  STRUCT
   FROM_MES_S702 : STRUCT
    STATION_MAIN : WORD ;
    DISTINCTION_LH_RH : WORD ;
    STAION_NUMBER : WORD ;
    BODY_TYPE_1ST : WORD ;
    BODY_TYPE_OPTION : WORD ;
    RBT1_STANDARD_WELD_DATA : WORD ;
    RBT2_STANDARD_WELD_DATA : WORD ;
    RBT3_STANDARD_WELD_DATA : WORD ;
    RBT4_STANDARD_WELD_DATA : WORD ;
    RBT5_STANDARD_WELD_DATA : WORD ;
    RBT6_STANDARD_WELD_DATA : WORD ;
    RBT7_STANDARD_WELD_DATA : WORD ;
    RBT8_STANDARD_WELD_DATA : WORD ;
    RBT9_STANDARD_WELD_DATA : WORD ;
    RBT10_STANDARD_WELD_DATA : WORD ;
    RBT11_STANDARD_WELD_DATA : WORD ;
    RBT12_STANDARD_WELD_DATA : WORD ;
    RBT13_STANDARD_WELD_DATA : WORD ;
    RBT14_STANDARD_WELD_DATA : WORD ;
    RBT15_STANDARD_WELD_DATA : WORD ;
    RBT16_STANDARD_WELD_DATA : WORD ;
    RBT17_STANDARD_WELD_DATA : WORD ;
    RBT18_STANDARD_WELD_DATA : WORD ;
    RBT19_STANDARD_WELD_DATA : WORD ;
    RBT20_STANDARD_WELD_DATA : WORD ;
    RBT21_STANDARD_WELD_DATA : WORD ;
    RBT22_STANDARD_WELD_DATA : WORD ;
    RBT23_STANDARD_WELD_DAT : WORD ;
    RBT24_STANDARD_WELD_DAT : WORD ;
    CHK_WORD : WORD ;
    TEST_TEMP : ARRAY  [1 .. 40 ] OF BYTE ;
   END_STRUCT ;
   FROM_MES_S703 : STRUCT
    STATION_MAIN : WORD ;
    DISTINCTION_LH_RH : WORD ;
    STAION_NUMBER : WORD ;
    BODY_TYPE_1ST : WORD ;
    BODY_TYPE_OPTION : WORD ;
    RBT1_STANDARD_WELD_DATA : WORD ;
    RBT2_STANDARD_WELD_DATA : WORD ;
    RBT3_STANDARD_WELD_DATA : WORD ;
    RBT4_STANDARD_WELD_DATA : WORD ;
    RBT5_STANDARD_WELD_DATA : WORD ;
    RBT6_STANDARD_WELD_DATA : WORD ;
    RBT7_STANDARD_WELD_DATA : WORD ;
    RBT8_STANDARD_WELD_DATA : WORD ;
    RBT9_STANDARD_WELD_DATA : WORD ;
    RBT10_STANDARD_WELD_DATA : WORD ;
    RBT11_STANDARD_WELD_DATA : WORD ;
    RBT12_STANDARD_WELD_DATA : WORD ;
    RBT13_STANDARD_WELD_DATA : WORD ;
    RBT14_STANDARD_WELD_DATA : WORD ;
    RBT15_STANDARD_WELD_DATA : WORD ;
    RBT16_STANDARD_WELD_DATA : WORD ;
    RBT17_STANDARD_WELD_DATA : WORD ;
    RBT18_STANDARD_WELD_DATA : WORD ;
    RBT19_STANDARD_WELD_DATA : WORD ;
    RBT20_STANDARD_WELD_DATA : WORD ;
    RBT21_STANDARD_WELD_DATA : WORD ;
    RBT22_STANDARD_WELD_DATA : WORD ;
    RBT23_STANDARD_WELD_DAT : WORD ;
    RBT24_STANDARD_WELD_DAT : WORD ;
    CHK_WORD : WORD ;
    TEST_TEMP : ARRAY  [1 .. 40 ] OF BYTE ;
   END_STRUCT ;
   FROM_MES_S704 : STRUCT
    STATION_MAIN : WORD ;
    DISTINCTION_LH_RH : WORD ;
    STAION_NUMBER : WORD ;
    BODY_TYPE_1ST : WORD ;
    BODY_TYPE_OPTION : WORD ;
    RBT1_STANDARD_WELD_DATA : WORD ;
    RBT2_STANDARD_WELD_DATA : WORD ;
    RBT3_STANDARD_WELD_DATA : WORD ;
    RBT4_STANDARD_WELD_DATA : WORD ;
    RBT5_STANDARD_WELD_DATA : WORD ;
    RBT6_STANDARD_WELD_DATA : WORD ;
    RBT7_STANDARD_WELD_DATA : WORD ;
    RBT8_STANDARD_WELD_DATA : WORD ;
    RBT9_STANDARD_WELD_DATA : WORD ;
    RBT10_STANDARD_WELD_DATA : WORD ;
    RBT11_STANDARD_WELD_DATA : WORD ;
    RBT12_STANDARD_WELD_DATA : WORD ;
    RBT13_STANDARD_WELD_DATA : WORD ;
    RBT14_STANDARD_WELD_DATA : WORD ;
    RBT15_STANDARD_WELD_DATA : WORD ;
    RBT16_STANDARD_WELD_DATA : WORD ;
    RBT17_STANDARD_WELD_DATA : WORD ;
    RBT18_STANDARD_WELD_DATA : WORD ;
    RBT19_STANDARD_WELD_DATA : WORD ;
    RBT20_STANDARD_WELD_DATA : WORD ;
    RBT21_STANDARD_WELD_DATA : WORD ;
    RBT22_STANDARD_WELD_DATA : WORD ;
    RBT23_STANDARD_WELD_DAT : WORD ;
    RBT24_STANDARD_WELD_DAT : WORD ;
    CHK_WORD : WORD ;
    TEST_TEMP : ARRAY  [1 .. 40 ] OF BYTE ;
   END_STRUCT ;
  END_STRUCT ;
BEGIN
   FROM_MES_S702.STATION_MAIN := W#16#0;
   FROM_MES_S702.DISTINCTION_LH_RH := W#16#0;
   FROM_MES_S702.STAION_NUMBER := W#16#0;
   FROM_MES_S702.BODY_TYPE_1ST := W#16#0;
   FROM_MES_S702.BODY_TYPE_OPTION := W#16#0;
   FROM_MES_S702.RBT1_STANDARD_WELD_DATA := W#16#0;
   FROM_MES_S702.RBT2_STANDARD_WELD_DATA := W#16#0;
   FROM_MES_S702.RBT3_STANDARD_WELD_DATA := W#16#0;
   FROM_MES_S702.RBT4_STANDARD_WELD_DATA := W#16#0;
   FROM_MES_S702.RBT5_STANDARD_WELD_DATA := W#16#0;
   FROM_MES_S702.RBT6_STANDARD_WELD_DATA := W#16#0;
   FROM_MES_S702.RBT7_STANDARD_WELD_DATA := W#16#0;
   FROM_MES_S702.RBT8_STANDARD_WELD_DATA := W#16#0;
   FROM_MES_S702.RBT9_STANDARD_WELD_DATA := W#16#0;
   FROM_MES_S702.RBT10_STANDARD_WELD_DATA := W#16#0;
   FROM_MES_S702.RBT11_STANDARD_WELD_DATA := W#16#0;
   FROM_MES_S702.RBT12_STANDARD_WELD_DATA := W#16#0;
   FROM_MES_S702.RBT13_STANDARD_WELD_DATA := W#16#0;
   FROM_MES_S702.RBT14_STANDARD_WELD_DATA := W#16#0;
   FROM_MES_S702.RBT15_STANDARD_WELD_DATA := W#16#0;
   FROM_MES_S702.RBT16_STANDARD_WELD_DATA := W#16#0;
   FROM_MES_S702.RBT17_STANDARD_WELD_DATA := W#16#0;
   FROM_MES_S702.RBT18_STANDARD_WELD_DATA := W#16#0;
   FROM_MES_S702.RBT19_STANDARD_WELD_DATA := W#16#0;
   FROM_MES_S702.RBT20_STANDARD_WELD_DATA := W#16#0;
   FROM_MES_S702.RBT21_STANDARD_WELD_DATA := W#16#0;
   FROM_MES_S702.RBT22_STANDARD_WELD_DATA := W#16#0;
   FROM_MES_S702.RBT23_STANDARD_WELD_DAT := W#16#0;
   FROM_MES_S702.RBT24_STANDARD_WELD_DAT := W#16#0;
   FROM_MES_S702.CHK_WORD := W#16#0;
   FROM_MES_S702.TEST_TEMP[1] := B#16#0;
   FROM_MES_S702.TEST_TEMP[2] := B#16#0;
   FROM_MES_S702.TEST_TEMP[3] := B#16#0;
   FROM_MES_S702.TEST_TEMP[4] := B#16#0;
   FROM_MES_S702.TEST_TEMP[5] := B#16#0;
   FROM_MES_S702.TEST_TEMP[6] := B#16#0;
   FROM_MES_S702.TEST_TEMP[7] := B#16#0;
   FROM_MES_S702.TEST_TEMP[8] := B#16#0;
   FROM_MES_S702.TEST_TEMP[9] := B#16#0;
   FROM_MES_S702.TEST_TEMP[10] := B#16#0;
   FROM_MES_S702.TEST_TEMP[11] := B#16#0;
   FROM_MES_S702.TEST_TEMP[12] := B#16#0;
   FROM_MES_S702.TEST_TEMP[13] := B#16#0;
   FROM_MES_S702.TEST_TEMP[14] := B#16#0;
   FROM_MES_S702.TEST_TEMP[15] := B#16#0;
   FROM_MES_S702.TEST_TEMP[16] := B#16#0;
   FROM_MES_S702.TEST_TEMP[17] := B#16#0;
   FROM_MES_S702.TEST_TEMP[18] := B#16#0;
   FROM_MES_S702.TEST_TEMP[19] := B#16#0;
   FROM_MES_S702.TEST_TEMP[20] := B#16#0;
   FROM_MES_S702.TEST_TEMP[21] := B#16#0;
   FROM_MES_S702.TEST_TEMP[22] := B#16#0;
   FROM_MES_S702.TEST_TEMP[23] := B#16#0;
   FROM_MES_S702.TEST_TEMP[24] := B#16#0;
   FROM_MES_S702.TEST_TEMP[25] := B#16#0;
   FROM_MES_S702.TEST_TEMP[26] := B#16#0;
   FROM_MES_S702.TEST_TEMP[27] := B#16#0;
   FROM_MES_S702.TEST_TEMP[28] := B#16#0;
   FROM_MES_S702.TEST_TEMP[29] := B#16#0;
   FROM_MES_S702.TEST_TEMP[30] := B#16#0;
   FROM_MES_S702.TEST_TEMP[31] := B#16#0;
   FROM_MES_S702.TEST_TEMP[32] := B#16#0;
   FROM_MES_S702.TEST_TEMP[33] := B#16#0;
   FROM_MES_S702.TEST_TEMP[34] := B#16#0;
   FROM_MES_S702.TEST_TEMP[35] := B#16#0;
   FROM_MES_S702.TEST_TEMP[36] := B#16#0;
   FROM_MES_S702.TEST_TEMP[37] := B#16#0;
   FROM_MES_S702.TEST_TEMP[38] := B#16#0;
   FROM_MES_S702.TEST_TEMP[39] := B#16#0;
   FROM_MES_S702.TEST_TEMP[40] := B#16#0;
   FROM_MES_S703.STATION_MAIN := W#16#0;
   FROM_MES_S703.DISTINCTION_LH_RH := W#16#0;
   FROM_MES_S703.STAION_NUMBER := W#16#0;
   FROM_MES_S703.BODY_TYPE_1ST := W#16#0;
   FROM_MES_S703.BODY_TYPE_OPTION := W#16#0;
   FROM_MES_S703.RBT1_STANDARD_WELD_DATA := W#16#0;
   FROM_MES_S703.RBT2_STANDARD_WELD_DATA := W#16#0;
   FROM_MES_S703.RBT3_STANDARD_WELD_DATA := W#16#0;
   FROM_MES_S703.RBT4_STANDARD_WELD_DATA := W#16#0;
   FROM_MES_S703.RBT5_STANDARD_WELD_DATA := W#16#0;
   FROM_MES_S703.RBT6_STANDARD_WELD_DATA := W#16#0;
   FROM_MES_S703.RBT7_STANDARD_WELD_DATA := W#16#0;
   FROM_MES_S703.RBT8_STANDARD_WELD_DATA := W#16#0;
   FROM_MES_S703.RBT9_STANDARD_WELD_DATA := W#16#0;
   FROM_MES_S703.RBT10_STANDARD_WELD_DATA := W#16#0;
   FROM_MES_S703.RBT11_STANDARD_WELD_DATA := W#16#0;
   FROM_MES_S703.RBT12_STANDARD_WELD_DATA := W#16#0;
   FROM_MES_S703.RBT13_STANDARD_WELD_DATA := W#16#0;
   FROM_MES_S703.RBT14_STANDARD_WELD_DATA := W#16#0;
   FROM_MES_S703.RBT15_STANDARD_WELD_DATA := W#16#0;
   FROM_MES_S703.RBT16_STANDARD_WELD_DATA := W#16#0;
   FROM_MES_S703.RBT17_STANDARD_WELD_DATA := W#16#0;
   FROM_MES_S703.RBT18_STANDARD_WELD_DATA := W#16#0;
   FROM_MES_S703.RBT19_STANDARD_WELD_DATA := W#16#0;
   FROM_MES_S703.RBT20_STANDARD_WELD_DATA := W#16#0;
   FROM_MES_S703.RBT21_STANDARD_WELD_DATA := W#16#0;
   FROM_MES_S703.RBT22_STANDARD_WELD_DATA := W#16#0;
   FROM_MES_S703.RBT23_STANDARD_WELD_DAT := W#16#0;
   FROM_MES_S703.RBT24_STANDARD_WELD_DAT := W#16#0;
   FROM_MES_S703.CHK_WORD := W#16#0;
   FROM_MES_S703.TEST_TEMP[1] := B#16#0;
   FROM_MES_S703.TEST_TEMP[2] := B#16#0;
   FROM_MES_S703.TEST_TEMP[3] := B#16#0;
   FROM_MES_S703.TEST_TEMP[4] := B#16#0;
   FROM_MES_S703.TEST_TEMP[5] := B#16#0;
   FROM_MES_S703.TEST_TEMP[6] := B#16#0;
   FROM_MES_S703.TEST_TEMP[7] := B#16#0;
   FROM_MES_S703.TEST_TEMP[8] := B#16#0;
   FROM_MES_S703.TEST_TEMP[9] := B#16#0;
   FROM_MES_S703.TEST_TEMP[10] := B#16#0;
   FROM_MES_S703.TEST_TEMP[11] := B#16#0;
   FROM_MES_S703.TEST_TEMP[12] := B#16#0;
   FROM_MES_S703.TEST_TEMP[13] := B#16#0;
   FROM_MES_S703.TEST_TEMP[14] := B#16#0;
   FROM_MES_S703.TEST_TEMP[15] := B#16#0;
   FROM_MES_S703.TEST_TEMP[16] := B#16#0;
   FROM_MES_S703.TEST_TEMP[17] := B#16#0;
   FROM_MES_S703.TEST_TEMP[18] := B#16#0;
   FROM_MES_S703.TEST_TEMP[19] := B#16#0;
   FROM_MES_S703.TEST_TEMP[20] := B#16#0;
   FROM_MES_S703.TEST_TEMP[21] := B#16#0;
   FROM_MES_S703.TEST_TEMP[22] := B#16#0;
   FROM_MES_S703.TEST_TEMP[23] := B#16#0;
   FROM_MES_S703.TEST_TEMP[24] := B#16#0;
   FROM_MES_S703.TEST_TEMP[25] := B#16#0;
   FROM_MES_S703.TEST_TEMP[26] := B#16#0;
   FROM_MES_S703.TEST_TEMP[27] := B#16#0;
   FROM_MES_S703.TEST_TEMP[28] := B#16#0;
   FROM_MES_S703.TEST_TEMP[29] := B#16#0;
   FROM_MES_S703.TEST_TEMP[30] := B#16#0;
   FROM_MES_S703.TEST_TEMP[31] := B#16#0;
   FROM_MES_S703.TEST_TEMP[32] := B#16#0;
   FROM_MES_S703.TEST_TEMP[33] := B#16#0;
   FROM_MES_S703.TEST_TEMP[34] := B#16#0;
   FROM_MES_S703.TEST_TEMP[35] := B#16#0;
   FROM_MES_S703.TEST_TEMP[36] := B#16#0;
   FROM_MES_S703.TEST_TEMP[37] := B#16#0;
   FROM_MES_S703.TEST_TEMP[38] := B#16#0;
   FROM_MES_S703.TEST_TEMP[39] := B#16#0;
   FROM_MES_S703.TEST_TEMP[40] := B#16#0;
   FROM_MES_S704.STATION_MAIN := W#16#0;
   FROM_MES_S704.DISTINCTION_LH_RH := W#16#0;
   FROM_MES_S704.STAION_NUMBER := W#16#0;
   FROM_MES_S704.BODY_TYPE_1ST := W#16#0;
   FROM_MES_S704.BODY_TYPE_OPTION := W#16#0;
   FROM_MES_S704.RBT1_STANDARD_WELD_DATA := W#16#0;
   FROM_MES_S704.RBT2_STANDARD_WELD_DATA := W#16#0;
   FROM_MES_S704.RBT3_STANDARD_WELD_DATA := W#16#0;
   FROM_MES_S704.RBT4_STANDARD_WELD_DATA := W#16#0;
   FROM_MES_S704.RBT5_STANDARD_WELD_DATA := W#16#0;
   FROM_MES_S704.RBT6_STANDARD_WELD_DATA := W#16#0;
   FROM_MES_S704.RBT7_STANDARD_WELD_DATA := W#16#0;
   FROM_MES_S704.RBT8_STANDARD_WELD_DATA := W#16#0;
   FROM_MES_S704.RBT9_STANDARD_WELD_DATA := W#16#0;
   FROM_MES_S704.RBT10_STANDARD_WELD_DATA := W#16#0;
   FROM_MES_S704.RBT11_STANDARD_WELD_DATA := W#16#0;
   FROM_MES_S704.RBT12_STANDARD_WELD_DATA := W#16#0;
   FROM_MES_S704.RBT13_STANDARD_WELD_DATA := W#16#0;
   FROM_MES_S704.RBT14_STANDARD_WELD_DATA := W#16#0;
   FROM_MES_S704.RBT15_STANDARD_WELD_DATA := W#16#0;
   FROM_MES_S704.RBT16_STANDARD_WELD_DATA := W#16#0;
   FROM_MES_S704.RBT17_STANDARD_WELD_DATA := W#16#0;
   FROM_MES_S704.RBT18_STANDARD_WELD_DATA := W#16#0;
   FROM_MES_S704.RBT19_STANDARD_WELD_DATA := W#16#0;
   FROM_MES_S704.RBT20_STANDARD_WELD_DATA := W#16#0;
   FROM_MES_S704.RBT21_STANDARD_WELD_DATA := W#16#0;
   FROM_MES_S704.RBT22_STANDARD_WELD_DATA := W#16#0;
   FROM_MES_S704.RBT23_STANDARD_WELD_DAT := W#16#0;
   FROM_MES_S704.RBT24_STANDARD_WELD_DAT := W#16#0;
   FROM_MES_S704.CHK_WORD := W#16#0;
   FROM_MES_S704.TEST_TEMP[1] := B#16#0;
   FROM_MES_S704.TEST_TEMP[2] := B#16#0;
   FROM_MES_S704.TEST_TEMP[3] := B#16#0;
   FROM_MES_S704.TEST_TEMP[4] := B#16#0;
   FROM_MES_S704.TEST_TEMP[5] := B#16#0;
   FROM_MES_S704.TEST_TEMP[6] := B#16#0;
   FROM_MES_S704.TEST_TEMP[7] := B#16#0;
   FROM_MES_S704.TEST_TEMP[8] := B#16#0;
   FROM_MES_S704.TEST_TEMP[9] := B#16#0;
   FROM_MES_S704.TEST_TEMP[10] := B#16#0;
   FROM_MES_S704.TEST_TEMP[11] := B#16#0;
   FROM_MES_S704.TEST_TEMP[12] := B#16#0;
   FROM_MES_S704.TEST_TEMP[13] := B#16#0;
   FROM_MES_S704.TEST_TEMP[14] := B#16#0;
   FROM_MES_S704.TEST_TEMP[15] := B#16#0;
   FROM_MES_S704.TEST_TEMP[16] := B#16#0;
   FROM_MES_S704.TEST_TEMP[17] := B#16#0;
   FROM_MES_S704.TEST_TEMP[18] := B#16#0;
   FROM_MES_S704.TEST_TEMP[19] := B#16#0;
   FROM_MES_S704.TEST_TEMP[20] := B#16#0;
   FROM_MES_S704.TEST_TEMP[21] := B#16#0;
   FROM_MES_S704.TEST_TEMP[22] := B#16#0;
   FROM_MES_S704.TEST_TEMP[23] := B#16#0;
   FROM_MES_S704.TEST_TEMP[24] := B#16#0;
   FROM_MES_S704.TEST_TEMP[25] := B#16#0;
   FROM_MES_S704.TEST_TEMP[26] := B#16#0;
   FROM_MES_S704.TEST_TEMP[27] := B#16#0;
   FROM_MES_S704.TEST_TEMP[28] := B#16#0;
   FROM_MES_S704.TEST_TEMP[29] := B#16#0;
   FROM_MES_S704.TEST_TEMP[30] := B#16#0;
   FROM_MES_S704.TEST_TEMP[31] := B#16#0;
   FROM_MES_S704.TEST_TEMP[32] := B#16#0;
   FROM_MES_S704.TEST_TEMP[33] := B#16#0;
   FROM_MES_S704.TEST_TEMP[34] := B#16#0;
   FROM_MES_S704.TEST_TEMP[35] := B#16#0;
   FROM_MES_S704.TEST_TEMP[36] := B#16#0;
   FROM_MES_S704.TEST_TEMP[37] := B#16#0;
   FROM_MES_S704.TEST_TEMP[38] := B#16#0;
   FROM_MES_S704.TEST_TEMP[39] := B#16#0;
   FROM_MES_S704.TEST_TEMP[40] := B#16#0;
END_DATA_BLOCK

DATA_BLOCK DB 41
TITLE =
VERSION : 0.1


  STRUCT
   S702_BT_CODE_2011 : STRUCT
    STATION_MAIN : WORD ;
    DISTINCTION_LH_RH : WORD ;
    STAION_NUMBER : WORD ;
    BODY_TYPE_1ST : WORD ;
    BODY_TYPE_OPTION : WORD ;
    RBT1_STANDARD_WELD_DATA : WORD ;
    RBT2_STANDARD_WELD_DATA : WORD ;
    RBT3_STANDARD_WELD_DATA : WORD ;
    RBT4_STANDARD_WELD_DATA : WORD ;
    RBT5_STANDARD_WELD_DATA : WORD ;
    RBT6_STANDARD_WELD_DATA : WORD ;
    RBT7_STANDARD_WELD_DATA : WORD ;
    RBT8_STANDARD_WELD_DATA : WORD ;
    RBT9_STANDARD_WELD_DATA : WORD ;
    RBT10_STANDARD_WELD_DATA : WORD ;
    RBT11_STANDARD_WELD_DATA : WORD ;
    RBT12_STANDARD_WELD_DATA : WORD ;
    RBT13_STANDARD_WELD_DATA : WORD ;
    RBT14_STANDARD_WELD_DATA : WORD ;
    RBT15_STANDARD_WELD_DATA : WORD ;
    RBT16_STANDARD_WELD_DATA : WORD ;
    RBT17_STANDARD_WELD_DATA : WORD ;
    RBT18_STANDARD_WELD_DATA : WORD ;
    RBT19_STANDARD_WELD_DATA : WORD ;
    RBT20_STANDARD_WELD_DATA : WORD ;
    RBT21_STANDARD_WELD_DATA : WORD ;
    RBT22_STANDARD_WELD_DATA : WORD ;
    RBT23_STANDARD_WELD_DAT : WORD ;
    RBT24_STANDARD_WELD_DAT : WORD ;
    CHK_WORD : WORD ;
    TEST_TEMP : ARRAY  [1 .. 40 ] OF BYTE ;
   END_STRUCT ;
   S702_BT_CODE_2012 : STRUCT
    STATION_MAIN : WORD ;
    DISTINCTION_LH_RH : WORD ;
    STAION_NUMBER : WORD ;
    BODY_TYPE_1ST : WORD ;
    BODY_TYPE_OPTION : WORD ;
    RBT1_STANDARD_WELD_DATA : WORD ;
    RBT2_STANDARD_WELD_DATA : WORD ;
    RBT3_STANDARD_WELD_DATA : WORD ;
    RBT4_STANDARD_WELD_DATA : WORD ;
    RBT5_STANDARD_WELD_DATA : WORD ;
    RBT6_STANDARD_WELD_DATA : WORD ;
    RBT7_STANDARD_WELD_DATA : WORD ;
    RBT8_STANDARD_WELD_DATA : WORD ;
    RBT9_STANDARD_WELD_DATA : WORD ;
    RBT10_STANDARD_WELD_DATA : WORD ;
    RBT11_STANDARD_WELD_DATA : WORD ;
    RBT12_STANDARD_WELD_DATA : WORD ;
    RBT13_STANDARD_WELD_DATA : WORD ;
    RBT14_STANDARD_WELD_DATA : WORD ;
    RBT15_STANDARD_WELD_DATA : WORD ;
    RBT16_STANDARD_WELD_DATA : WORD ;
    RBT17_STANDARD_WELD_DATA : WORD ;
    RBT18_STANDARD_WELD_DATA : WORD ;
    RBT19_STANDARD_WELD_DATA : WORD ;
    RBT20_STANDARD_WELD_DATA : WORD ;
    RBT21_STANDARD_WELD_DATA : WORD ;
    RBT22_STANDARD_WELD_DATA : WORD ;
    RBT23_STANDARD_WELD_DAT : WORD ;
    RBT24_STANDARD_WELD_DAT : WORD ;
    CHK_WORD : WORD ;
    TEST_TEMP : ARRAY  [1 .. 40 ] OF BYTE ;
   END_STRUCT ;
   S702_BT_CODE_2013 : STRUCT
    STATION_MAIN : WORD ;
    DISTINCTION_LH_RH : WORD ;
    STAION_NUMBER : WORD ;
    BODY_TYPE_1ST : WORD ;
    BODY_TYPE_OPTION : WORD ;
    RBT1_STANDARD_WELD_DATA : WORD ;
    RBT2_STANDARD_WELD_DATA : WORD ;
    RBT3_STANDARD_WELD_DATA : WORD ;
    RBT4_STANDARD_WELD_DATA : WORD ;
    RBT5_STANDARD_WELD_DATA : WORD ;
    RBT6_STANDARD_WELD_DATA : WORD ;
    RBT7_STANDARD_WELD_DATA : WORD ;
    RBT8_STANDARD_WELD_DATA : WORD ;
    RBT9_STANDARD_WELD_DATA : WORD ;
    RBT10_STANDARD_WELD_DATA : WORD ;
    RBT11_STANDARD_WELD_DATA : WORD ;
    RBT12_STANDARD_WELD_DATA : WORD ;
    RBT13_STANDARD_WELD_DATA : WORD ;
    RBT14_STANDARD_WELD_DATA : WORD ;
    RBT15_STANDARD_WELD_DATA : WORD ;
    RBT16_STANDARD_WELD_DATA : WORD ;
    RBT17_STANDARD_WELD_DATA : WORD ;
    RBT18_STANDARD_WELD_DATA : WORD ;
    RBT19_STANDARD_WELD_DATA : WORD ;
    RBT20_STANDARD_WELD_DATA : WORD ;
    RBT21_STANDARD_WELD_DATA : WORD ;
    RBT22_STANDARD_WELD_DATA : WORD ;
    RBT23_STANDARD_WELD_DAT : WORD ;
    RBT24_STANDARD_WELD_DAT : WORD ;
    CHK_WORD : WORD ;
    TEST_TEMP : ARRAY  [1 .. 40 ] OF BYTE ;
   END_STRUCT ;
   S702_BT_CODE_2014 : STRUCT
    STATION_MAIN : WORD ;
    DISTINCTION_LH_RH : WORD ;
    STAION_NUMBER : WORD ;
    BODY_TYPE_1ST : WORD ;
    BODY_TYPE_OPTION : WORD ;
    RBT1_STANDARD_WELD_DATA : WORD ;
    RBT2_STANDARD_WELD_DATA : WORD ;
    RBT3_STANDARD_WELD_DATA : WORD ;
    RBT4_STANDARD_WELD_DATA : WORD ;
    RBT5_STANDARD_WELD_DATA : WORD ;
    RBT6_STANDARD_WELD_DATA : WORD ;
    RBT7_STANDARD_WELD_DATA : WORD ;
    RBT8_STANDARD_WELD_DATA : WORD ;
    RBT9_STANDARD_WELD_DATA : WORD ;
    RBT10_STANDARD_WELD_DATA : WORD ;
    RBT11_STANDARD_WELD_DATA : WORD ;
    RBT12_STANDARD_WELD_DATA : WORD ;
    RBT13_STANDARD_WELD_DATA : WORD ;
    RBT14_STANDARD_WELD_DATA : WORD ;
    RBT15_STANDARD_WELD_DATA : WORD ;
    RBT16_STANDARD_WELD_DATA : WORD ;
    RBT17_STANDARD_WELD_DATA : WORD ;
    RBT18_STANDARD_WELD_DATA : WORD ;
    RBT19_STANDARD_WELD_DATA : WORD ;
    RBT20_STANDARD_WELD_DATA : WORD ;
    RBT21_STANDARD_WELD_DATA : WORD ;
    RBT22_STANDARD_WELD_DATA : WORD ;
    RBT23_STANDARD_WELD_DAT : WORD ;
    RBT24_STANDARD_WELD_DAT : WORD ;
    CHK_WORD : WORD ;
    TEST_TEMP : ARRAY  [1 .. 40 ] OF BYTE ;
   END_STRUCT ;
   S702_BT_CODE_2015 : STRUCT
    STATION_MAIN : WORD ;
    DISTINCTION_LH_RH : WORD ;
    STAION_NUMBER : WORD ;
    BODY_TYPE_1ST : WORD ;
    BODY_TYPE_OPTION : WORD ;
    RBT1_STANDARD_WELD_DATA : WORD ;
    RBT2_STANDARD_WELD_DATA : WORD ;
    RBT3_STANDARD_WELD_DATA : WORD ;
    RBT4_STANDARD_WELD_DATA : WORD ;
    RBT5_STANDARD_WELD_DATA : WORD ;
    RBT6_STANDARD_WELD_DATA : WORD ;
    RBT7_STANDARD_WELD_DATA : WORD ;
    RBT8_STANDARD_WELD_DATA : WORD ;
    RBT9_STANDARD_WELD_DATA : WORD ;
    RBT10_STANDARD_WELD_DATA : WORD ;
    RBT11_STANDARD_WELD_DATA : WORD ;
    RBT12_STANDARD_WELD_DATA : WORD ;
    RBT13_STANDARD_WELD_DATA : WORD ;
    RBT14_STANDARD_WELD_DATA : WORD ;
    RBT15_STANDARD_WELD_DATA : WORD ;
    RBT16_STANDARD_WELD_DATA : WORD ;
    RBT17_STANDARD_WELD_DATA : WORD ;
    RBT18_STANDARD_WELD_DATA : WORD ;
    RBT19_STANDARD_WELD_DATA : WORD ;
    RBT20_STANDARD_WELD_DATA : WORD ;
    RBT21_STANDARD_WELD_DATA : WORD ;
    RBT22_STANDARD_WELD_DATA : WORD ;
    RBT23_STANDARD_WELD_DAT : WORD ;
    RBT24_STANDARD_WELD_DAT : WORD ;
    CHK_WORD : WORD ;
    TEST_TEMP : ARRAY  [1 .. 40 ] OF BYTE ;
   END_STRUCT ;
   S702_BT_CODE_2016 : STRUCT
    STATION_MAIN : WORD ;
    DISTINCTION_LH_RH : WORD ;
    STAION_NUMBER : WORD ;
    BODY_TYPE_1ST : WORD ;
    BODY_TYPE_OPTION : WORD ;
    RBT1_STANDARD_WELD_DATA : WORD ;
    RBT2_STANDARD_WELD_DATA : WORD ;
    RBT3_STANDARD_WELD_DATA : WORD ;
    RBT4_STANDARD_WELD_DATA : WORD ;
    RBT5_STANDARD_WELD_DATA : WORD ;
    RBT6_STANDARD_WELD_DATA : WORD ;
    RBT7_STANDARD_WELD_DATA : WORD ;
    RBT8_STANDARD_WELD_DATA : WORD ;
    RBT9_STANDARD_WELD_DATA : WORD ;
    RBT10_STANDARD_WELD_DATA : WORD ;
    RBT11_STANDARD_WELD_DATA : WORD ;
    RBT12_STANDARD_WELD_DATA : WORD ;
    RBT13_STANDARD_WELD_DATA : WORD ;
    RBT14_STANDARD_WELD_DATA : WORD ;
    RBT15_STANDARD_WELD_DATA : WORD ;
    RBT16_STANDARD_WELD_DATA : WORD ;
    RBT17_STANDARD_WELD_DATA : WORD ;
    RBT18_STANDARD_WELD_DATA : WORD ;
    RBT19_STANDARD_WELD_DATA : WORD ;
    RBT20_STANDARD_WELD_DATA : WORD ;
    RBT21_STANDARD_WELD_DATA : WORD ;
    RBT22_STANDARD_WELD_DATA : WORD ;
    RBT23_STANDARD_WELD_DAT : WORD ;
    RBT24_STANDARD_WELD_DAT : WORD ;
    CHK_WORD : WORD ;
    TEST_TEMP : ARRAY  [1 .. 40 ] OF BYTE ;
   END_STRUCT ;
   S702_BT_CODE_2017 : STRUCT
    STATION_MAIN : WORD ;
    DISTINCTION_LH_RH : WORD ;
    STAION_NUMBER : WORD ;
    BODY_TYPE_1ST : WORD ;
    BODY_TYPE_OPTION : WORD ;
    RBT1_STANDARD_WELD_DATA : WORD ;
    RBT2_STANDARD_WELD_DATA : WORD ;
    RBT3_STANDARD_WELD_DATA : WORD ;
    RBT4_STANDARD_WELD_DATA : WORD ;
    RBT5_STANDARD_WELD_DATA : WORD ;
    RBT6_STANDARD_WELD_DATA : WORD ;
    RBT7_STANDARD_WELD_DATA : WORD ;
    RBT8_STANDARD_WELD_DATA : WORD ;
    RBT9_STANDARD_WELD_DATA : WORD ;
    RBT10_STANDARD_WELD_DATA : WORD ;
    RBT11_STANDARD_WELD_DATA : WORD ;
    RBT12_STANDARD_WELD_DATA : WORD ;
    RBT13_STANDARD_WELD_DATA : WORD ;
    RBT14_STANDARD_WELD_DATA : WORD ;
    RBT15_STANDARD_WELD_DATA : WORD ;
    RBT16_STANDARD_WELD_DATA : WORD ;
    RBT17_STANDARD_WELD_DATA : WORD ;
    RBT18_STANDARD_WELD_DATA : WORD ;
    RBT19_STANDARD_WELD_DATA : WORD ;
    RBT20_STANDARD_WELD_DATA : WORD ;
    RBT21_STANDARD_WELD_DATA : WORD ;
    RBT22_STANDARD_WELD_DATA : WORD ;
    RBT23_STANDARD_WELD_DAT : WORD ;
    RBT24_STANDARD_WELD_DAT : WORD ;
    CHK_WORD : WORD ;
    TEST_TEMP : ARRAY  [1 .. 40 ] OF BYTE ;
   END_STRUCT ;
   S702_BT_CODE_2018 : STRUCT
    STATION_MAIN : WORD ;
    DISTINCTION_LH_RH : WORD ;
    STAION_NUMBER : WORD ;
    BODY_TYPE_1ST : WORD ;
    BODY_TYPE_OPTION : WORD ;
    RBT1_STANDARD_WELD_DATA : WORD ;
    RBT2_STANDARD_WELD_DATA : WORD ;
    RBT3_STANDARD_WELD_DATA : WORD ;
    RBT4_STANDARD_WELD_DATA : WORD ;
    RBT5_STANDARD_WELD_DATA : WORD ;
    RBT6_STANDARD_WELD_DATA : WORD ;
    RBT7_STANDARD_WELD_DATA : WORD ;
    RBT8_STANDARD_WELD_DATA : WORD ;
    RBT9_STANDARD_WELD_DATA : WORD ;
    RBT10_STANDARD_WELD_DATA : WORD ;
    RBT11_STANDARD_WELD_DATA : WORD ;
    RBT12_STANDARD_WELD_DATA : WORD ;
    RBT13_STANDARD_WELD_DATA : WORD ;
    RBT14_STANDARD_WELD_DATA : WORD ;
    RBT15_STANDARD_WELD_DATA : WORD ;
    RBT16_STANDARD_WELD_DATA : WORD ;
    RBT17_STANDARD_WELD_DATA : WORD ;
    RBT18_STANDARD_WELD_DATA : WORD ;
    RBT19_STANDARD_WELD_DATA : WORD ;
    RBT20_STANDARD_WELD_DATA : WORD ;
    RBT21_STANDARD_WELD_DATA : WORD ;
    RBT22_STANDARD_WELD_DATA : WORD ;
    RBT23_STANDARD_WELD_DAT : WORD ;
    RBT24_STANDARD_WELD_DAT : WORD ;
    CHK_WORD : WORD ;
    TEST_TEMP : ARRAY  [1 .. 40 ] OF BYTE ;
   END_STRUCT ;
   S702_BT_CODE_2019 : STRUCT
    STATION_MAIN : WORD ;
    DISTINCTION_LH_RH : WORD ;
    STAION_NUMBER : WORD ;
    BODY_TYPE_1ST : WORD ;
    BODY_TYPE_OPTION : WORD ;
    RBT1_STANDARD_WELD_DATA : WORD ;
    RBT2_STANDARD_WELD_DATA : WORD ;
    RBT3_STANDARD_WELD_DATA : WORD ;
    RBT4_STANDARD_WELD_DATA : WORD ;
    RBT5_STANDARD_WELD_DATA : WORD ;
    RBT6_STANDARD_WELD_DATA : WORD ;
    RBT7_STANDARD_WELD_DATA : WORD ;
    RBT8_STANDARD_WELD_DATA : WORD ;
    RBT9_STANDARD_WELD_DATA : WORD ;
    RBT10_STANDARD_WELD_DATA : WORD ;
    RBT11_STANDARD_WELD_DATA : WORD ;
    RBT12_STANDARD_WELD_DATA : WORD ;
    RBT13_STANDARD_WELD_DATA : WORD ;
    RBT14_STANDARD_WELD_DATA : WORD ;
    RBT15_STANDARD_WELD_DATA : WORD ;
    RBT16_STANDARD_WELD_DATA : WORD ;
    RBT17_STANDARD_WELD_DATA : WORD ;
    RBT18_STANDARD_WELD_DATA : WORD ;
    RBT19_STANDARD_WELD_DATA : WORD ;
    RBT20_STANDARD_WELD_DATA : WORD ;
    RBT21_STANDARD_WELD_DATA : WORD ;
    RBT22_STANDARD_WELD_DATA : WORD ;
    RBT23_STANDARD_WELD_DAT : WORD ;
    RBT24_STANDARD_WELD_DAT : WORD ;
    CHK_WORD : WORD ;
    TEST_TEMP : ARRAY  [1 .. 40 ] OF BYTE ;
   END_STRUCT ;
   S702_BT_CODE_2020 : STRUCT
    STATION_MAIN : WORD ;
    DISTINCTION_LH_RH : WORD ;
    STAION_NUMBER : WORD ;
    BODY_TYPE_1ST : WORD ;
    BODY_TYPE_OPTION : WORD ;
    RBT1_STANDARD_WELD_DATA : WORD ;
    RBT2_STANDARD_WELD_DATA : WORD ;
    RBT3_STANDARD_WELD_DATA : WORD ;
    RBT4_STANDARD_WELD_DATA : WORD ;
    RBT5_STANDARD_WELD_DATA : WORD ;
    RBT6_STANDARD_WELD_DATA : WORD ;
    RBT7_STANDARD_WELD_DATA : WORD ;
    RBT8_STANDARD_WELD_DATA : WORD ;
    RBT9_STANDARD_WELD_DATA : WORD ;
    RBT10_STANDARD_WELD_DATA : WORD ;
    RBT11_STANDARD_WELD_DATA : WORD ;
    RBT12_STANDARD_WELD_DATA : WORD ;
    RBT13_STANDARD_WELD_DATA : WORD ;
    RBT14_STANDARD_WELD_DATA : WORD ;
    RBT15_STANDARD_WELD_DATA : WORD ;
    RBT16_STANDARD_WELD_DATA : WORD ;
    RBT17_STANDARD_WELD_DATA : WORD ;
    RBT18_STANDARD_WELD_DATA : WORD ;
    RBT19_STANDARD_WELD_DATA : WORD ;
    RBT20_STANDARD_WELD_DATA : WORD ;
    RBT21_STANDARD_WELD_DATA : WORD ;
    RBT22_STANDARD_WELD_DATA : WORD ;
    RBT23_STANDARD_WELD_DAT : WORD ;
    RBT24_STANDARD_WELD_DAT : WORD ;
    CHK_WORD : WORD ;
    TEST_TEMP : ARRAY  [1 .. 40 ] OF BYTE ;
   END_STRUCT ;
   S702_BT_CODE_2021 : STRUCT
    STATION_MAIN : WORD ;
    DISTINCTION_LH_RH : WORD ;
    STAION_NUMBER : WORD ;
    BODY_TYPE_1ST : WORD ;
    BODY_TYPE_OPTION : WORD ;
    RBT1_STANDARD_WELD_DATA : WORD ;
    RBT2_STANDARD_WELD_DATA : WORD ;
    RBT3_STANDARD_WELD_DATA : WORD ;
    RBT4_STANDARD_WELD_DATA : WORD ;
    RBT5_STANDARD_WELD_DATA : WORD ;
    RBT6_STANDARD_WELD_DATA : WORD ;
    RBT7_STANDARD_WELD_DATA : WORD ;
    RBT8_STANDARD_WELD_DATA : WORD ;
    RBT9_STANDARD_WELD_DATA : WORD ;
    RBT10_STANDARD_WELD_DATA : WORD ;
    RBT11_STANDARD_WELD_DATA : WORD ;
    RBT12_STANDARD_WELD_DATA : WORD ;
    RBT13_STANDARD_WELD_DATA : WORD ;
    RBT14_STANDARD_WELD_DATA : WORD ;
    RBT15_STANDARD_WELD_DATA : WORD ;
    RBT16_STANDARD_WELD_DATA : WORD ;
    RBT17_STANDARD_WELD_DATA : WORD ;
    RBT18_STANDARD_WELD_DATA : WORD ;
    RBT19_STANDARD_WELD_DATA : WORD ;
    RBT20_STANDARD_WELD_DATA : WORD ;
    RBT21_STANDARD_WELD_DATA : WORD ;
    RBT22_STANDARD_WELD_DATA : WORD ;
    RBT23_STANDARD_WELD_DAT : WORD ;
    RBT24_STANDARD_WELD_DAT : WORD ;
    CHK_WORD : WORD ;
    TEST_TEMP : ARRAY  [1 .. 40 ] OF BYTE ;
   END_STRUCT ;
   S702_BT_CODE_2022 : STRUCT
    STATION_MAIN : WORD ;
    DISTINCTION_LH_RH : WORD ;
    STAION_NUMBER : WORD ;
    BODY_TYPE_1ST : WORD ;
    BODY_TYPE_OPTION : WORD ;
    RBT1_STANDARD_WELD_DATA : WORD ;
    RBT2_STANDARD_WELD_DATA : WORD ;
    RBT3_STANDARD_WELD_DATA : WORD ;
    RBT4_STANDARD_WELD_DATA : WORD ;
    RBT5_STANDARD_WELD_DATA : WORD ;
    RBT6_STANDARD_WELD_DATA : WORD ;
    RBT7_STANDARD_WELD_DATA : WORD ;
    RBT8_STANDARD_WELD_DATA : WORD ;
    RBT9_STANDARD_WELD_DATA : WORD ;
    RBT10_STANDARD_WELD_DATA : WORD ;
    RBT11_STANDARD_WELD_DATA : WORD ;
    RBT12_STANDARD_WELD_DATA : WORD ;
    RBT13_STANDARD_WELD_DATA : WORD ;
    RBT14_STANDARD_WELD_DATA : WORD ;
    RBT15_STANDARD_WELD_DATA : WORD ;
    RBT16_STANDARD_WELD_DATA : WORD ;
    RBT17_STANDARD_WELD_DATA : WORD ;
    RBT18_STANDARD_WELD_DATA : WORD ;
    RBT19_STANDARD_WELD_DATA : WORD ;
    RBT20_STANDARD_WELD_DATA : WORD ;
    RBT21_STANDARD_WELD_DATA : WORD ;
    RBT22_STANDARD_WELD_DATA : WORD ;
    RBT23_STANDARD_WELD_DAT : WORD ;
    RBT24_STANDARD_WELD_DAT : WORD ;
    CHK_WORD : WORD ;
    TEST_TEMP : ARRAY  [1 .. 40 ] OF BYTE ;
   END_STRUCT ;
   S702_BT_CODE_2023 : STRUCT
    STATION_MAIN : WORD ;
    DISTINCTION_LH_RH : WORD ;
    STAION_NUMBER : WORD ;
    BODY_TYPE_1ST : WORD ;
    BODY_TYPE_OPTION : WORD ;
    RBT1_STANDARD_WELD_DATA : WORD ;
    RBT2_STANDARD_WELD_DATA : WORD ;
    RBT3_STANDARD_WELD_DATA : WORD ;
    RBT4_STANDARD_WELD_DATA : WORD ;
    RBT5_STANDARD_WELD_DATA : WORD ;
    RBT6_STANDARD_WELD_DATA : WORD ;
    RBT7_STANDARD_WELD_DATA : WORD ;
    RBT8_STANDARD_WELD_DATA : WORD ;
    RBT9_STANDARD_WELD_DATA : WORD ;
    RBT10_STANDARD_WELD_DATA : WORD ;
    RBT11_STANDARD_WELD_DATA : WORD ;
    RBT12_STANDARD_WELD_DATA : WORD ;
    RBT13_STANDARD_WELD_DATA : WORD ;
    RBT14_STANDARD_WELD_DATA : WORD ;
    RBT15_STANDARD_WELD_DATA : WORD ;
    RBT16_STANDARD_WELD_DATA : WORD ;
    RBT17_STANDARD_WELD_DATA : WORD ;
    RBT18_STANDARD_WELD_DATA : WORD ;
    RBT19_STANDARD_WELD_DATA : WORD ;
    RBT20_STANDARD_WELD_DATA : WORD ;
    RBT21_STANDARD_WELD_DATA : WORD ;
    RBT22_STANDARD_WELD_DATA : WORD ;
    RBT23_STANDARD_WELD_DAT : WORD ;
    RBT24_STANDARD_WELD_DAT : WORD ;
    CHK_WORD : WORD ;
    TEST_TEMP : ARRAY  [1 .. 40 ] OF BYTE ;
   END_STRUCT ;
   S702_BT_CODE_2024 : STRUCT
    STATION_MAIN : WORD ;
    DISTINCTION_LH_RH : WORD ;
    STAION_NUMBER : WORD ;
    BODY_TYPE_1ST : WORD ;
    BODY_TYPE_OPTION : WORD ;
    RBT1_STANDARD_WELD_DATA : WORD ;
    RBT2_STANDARD_WELD_DATA : WORD ;
    RBT3_STANDARD_WELD_DATA : WORD ;
    RBT4_STANDARD_WELD_DATA : WORD ;
    RBT5_STANDARD_WELD_DATA : WORD ;
    RBT6_STANDARD_WELD_DATA : WORD ;
    RBT7_STANDARD_WELD_DATA : WORD ;
    RBT8_STANDARD_WELD_DATA : WORD ;
    RBT9_STANDARD_WELD_DATA : WORD ;
    RBT10_STANDARD_WELD_DATA : WORD ;
    RBT11_STANDARD_WELD_DATA : WORD ;
    RBT12_STANDARD_WELD_DATA : WORD ;
    RBT13_STANDARD_WELD_DATA : WORD ;
    RBT14_STANDARD_WELD_DATA : WORD ;
    RBT15_STANDARD_WELD_DATA : WORD ;
    RBT16_STANDARD_WELD_DATA : WORD ;
    RBT17_STANDARD_WELD_DATA : WORD ;
    RBT18_STANDARD_WELD_DATA : WORD ;
    RBT19_STANDARD_WELD_DATA : WORD ;
    RBT20_STANDARD_WELD_DATA : WORD ;
    RBT21_STANDARD_WELD_DATA : WORD ;
    RBT22_STANDARD_WELD_DATA : WORD ;
    RBT23_STANDARD_WELD_DAT : WORD ;
    RBT24_STANDARD_WELD_DAT : WORD ;
    CHK_WORD : WORD ;
    TEST_TEMP : ARRAY  [1 .. 40 ] OF BYTE ;
   END_STRUCT ;
   S702_BT_CODE_2025 : STRUCT
    STATION_MAIN : WORD ;
    DISTINCTION_LH_RH : WORD ;
    STAION_NUMBER : WORD ;
    BODY_TYPE_1ST : WORD ;
    BODY_TYPE_OPTION : WORD ;
    RBT1_STANDARD_WELD_DATA : WORD ;
    RBT2_STANDARD_WELD_DATA : WORD ;
    RBT3_STANDARD_WELD_DATA : WORD ;
    RBT4_STANDARD_WELD_DATA : WORD ;
    RBT5_STANDARD_WELD_DATA : WORD ;
    RBT6_STANDARD_WELD_DATA : WORD ;
    RBT7_STANDARD_WELD_DATA : WORD ;
    RBT8_STANDARD_WELD_DATA : WORD ;
    RBT9_STANDARD_WELD_DATA : WORD ;
    RBT10_STANDARD_WELD_DATA : WORD ;
    RBT11_STANDARD_WELD_DATA : WORD ;
    RBT12_STANDARD_WELD_DATA : WORD ;
    RBT13_STANDARD_WELD_DATA : WORD ;
    RBT14_STANDARD_WELD_DATA : WORD ;
    RBT15_STANDARD_WELD_DATA : WORD ;
    RBT16_STANDARD_WELD_DATA : WORD ;
    RBT17_STANDARD_WELD_DATA : WORD ;
    RBT18_STANDARD_WELD_DATA : WORD ;
    RBT19_STANDARD_WELD_DATA : WORD ;
    RBT20_STANDARD_WELD_DATA : WORD ;
    RBT21_STANDARD_WELD_DATA : WORD ;
    RBT22_STANDARD_WELD_DATA : WORD ;
    RBT23_STANDARD_WELD_DAT : WORD ;
    RBT24_STANDARD_WELD_DAT : WORD ;
    CHK_WORD : WORD ;
    TEST_TEMP : ARRAY  [1 .. 40 ] OF BYTE ;
   END_STRUCT ;
   S702_BT_CODE_2026 : STRUCT
    STATION_MAIN : WORD ;
    DISTINCTION_LH_RH : WORD ;
    STAION_NUMBER : WORD ;
    BODY_TYPE_1ST : WORD ;
    BODY_TYPE_OPTION : WORD ;
    RBT1_STANDARD_WELD_DATA : WORD ;
    RBT2_STANDARD_WELD_DATA : WORD ;
    RBT3_STANDARD_WELD_DATA : WORD ;
    RBT4_STANDARD_WELD_DATA : WORD ;
    RBT5_STANDARD_WELD_DATA : WORD ;
    RBT6_STANDARD_WELD_DATA : WORD ;
    RBT7_STANDARD_WELD_DATA : WORD ;
    RBT8_STANDARD_WELD_DATA : WORD ;
    RBT9_STANDARD_WELD_DATA : WORD ;
    RBT10_STANDARD_WELD_DATA : WORD ;
    RBT11_STANDARD_WELD_DATA : WORD ;
    RBT12_STANDARD_WELD_DATA : WORD ;
    RBT13_STANDARD_WELD_DATA : WORD ;
    RBT14_STANDARD_WELD_DATA : WORD ;
    RBT15_STANDARD_WELD_DATA : WORD ;
    RBT16_STANDARD_WELD_DATA : WORD ;
    RBT17_STANDARD_WELD_DATA : WORD ;
    RBT18_STANDARD_WELD_DATA : WORD ;
    RBT19_STANDARD_WELD_DATA : WORD ;
    RBT20_STANDARD_WELD_DATA : WORD ;
    RBT21_STANDARD_WELD_DATA : WORD ;
    RBT22_STANDARD_WELD_DATA : WORD ;
    RBT23_STANDARD_WELD_DAT : WORD ;
    RBT24_STANDARD_WELD_DAT : WORD ;
    CHK_WORD : WORD ;
    TEST_TEMP : ARRAY  [1 .. 40 ] OF BYTE ;
   END_STRUCT ;
   S702_BT_CODE_2027 : STRUCT
    STATION_MAIN : WORD ;
    DISTINCTION_LH_RH : WORD ;
    STAION_NUMBER : WORD ;
    BODY_TYPE_1ST : WORD ;
    BODY_TYPE_OPTION : WORD ;
    RBT1_STANDARD_WELD_DATA : WORD ;
    RBT2_STANDARD_WELD_DATA : WORD ;
    RBT3_STANDARD_WELD_DATA : WORD ;
    RBT4_STANDARD_WELD_DATA : WORD ;
    RBT5_STANDARD_WELD_DATA : WORD ;
    RBT6_STANDARD_WELD_DATA : WORD ;
    RBT7_STANDARD_WELD_DATA : WORD ;
    RBT8_STANDARD_WELD_DATA : WORD ;
    RBT9_STANDARD_WELD_DATA : WORD ;
    RBT10_STANDARD_WELD_DATA : WORD ;
    RBT11_STANDARD_WELD_DATA : WORD ;
    RBT12_STANDARD_WELD_DATA : WORD ;
    RBT13_STANDARD_WELD_DATA : WORD ;
    RBT14_STANDARD_WELD_DATA : WORD ;
    RBT15_STANDARD_WELD_DATA : WORD ;
    RBT16_STANDARD_WELD_DATA : WORD ;
    RBT17_STANDARD_WELD_DATA : WORD ;
    RBT18_STANDARD_WELD_DATA : WORD ;
    RBT19_STANDARD_WELD_DATA : WORD ;
    RBT20_STANDARD_WELD_DATA : WORD ;
    RBT21_STANDARD_WELD_DATA : WORD ;
    RBT22_STANDARD_WELD_DATA : WORD ;
    RBT23_STANDARD_WELD_DAT : WORD ;
    RBT24_STANDARD_WELD_DAT : WORD ;
    CHK_WORD : WORD ;
    TEST_TEMP : ARRAY  [1 .. 40 ] OF BYTE ;
   END_STRUCT ;
   S702_BT_CODE_2028 : STRUCT
    STATION_MAIN : WORD ;
    DISTINCTION_LH_RH : WORD ;
    STAION_NUMBER : WORD ;
    BODY_TYPE_1ST : WORD ;
    BODY_TYPE_OPTION : WORD ;
    RBT1_STANDARD_WELD_DATA : WORD ;
    RBT2_STANDARD_WELD_DATA : WORD ;
    RBT3_STANDARD_WELD_DATA : WORD ;
    RBT4_STANDARD_WELD_DATA : WORD ;
    RBT5_STANDARD_WELD_DATA : WORD ;
    RBT6_STANDARD_WELD_DATA : WORD ;
    RBT7_STANDARD_WELD_DATA : WORD ;
    RBT8_STANDARD_WELD_DATA : WORD ;
    RBT9_STANDARD_WELD_DATA : WORD ;
    RBT10_STANDARD_WELD_DATA : WORD ;
    RBT11_STANDARD_WELD_DATA : WORD ;
    RBT12_STANDARD_WELD_DATA : WORD ;
    RBT13_STANDARD_WELD_DATA : WORD ;
    RBT14_STANDARD_WELD_DATA : WORD ;
    RBT15_STANDARD_WELD_DATA : WORD ;
    RBT16_STANDARD_WELD_DATA : WORD ;
    RBT17_STANDARD_WELD_DATA : WORD ;
    RBT18_STANDARD_WELD_DATA : WORD ;
    RBT19_STANDARD_WELD_DATA : WORD ;
    RBT20_STANDARD_WELD_DATA : WORD ;
    RBT21_STANDARD_WELD_DATA : WORD ;
    RBT22_STANDARD_WELD_DATA : WORD ;
    RBT23_STANDARD_WELD_DAT : WORD ;
    RBT24_STANDARD_WELD_DAT : WORD ;
    CHK_WORD : WORD ;
    TEST_TEMP : ARRAY  [1 .. 40 ] OF BYTE ;
   END_STRUCT ;
   S702_BT_CODE_2029 : STRUCT
    STATION_MAIN : WORD ;
    DISTINCTION_LH_RH : WORD ;
    STAION_NUMBER : WORD ;
    BODY_TYPE_1ST : WORD ;
    BODY_TYPE_OPTION : WORD ;
    RBT1_STANDARD_WELD_DATA : WORD ;
    RBT2_STANDARD_WELD_DATA : WORD ;
    RBT3_STANDARD_WELD_DATA : WORD ;
    RBT4_STANDARD_WELD_DATA : WORD ;
    RBT5_STANDARD_WELD_DATA : WORD ;
    RBT6_STANDARD_WELD_DATA : WORD ;
    RBT7_STANDARD_WELD_DATA : WORD ;
    RBT8_STANDARD_WELD_DATA : WORD ;
    RBT9_STANDARD_WELD_DATA : WORD ;
    RBT10_STANDARD_WELD_DATA : WORD ;
    RBT11_STANDARD_WELD_DATA : WORD ;
    RBT12_STANDARD_WELD_DATA : WORD ;
    RBT13_STANDARD_WELD_DATA : WORD ;
    RBT14_STANDARD_WELD_DATA : WORD ;
    RBT15_STANDARD_WELD_DATA : WORD ;
    RBT16_STANDARD_WELD_DATA : WORD ;
    RBT17_STANDARD_WELD_DATA : WORD ;
    RBT18_STANDARD_WELD_DATA : WORD ;
    RBT19_STANDARD_WELD_DATA : WORD ;
    RBT20_STANDARD_WELD_DATA : WORD ;
    RBT21_STANDARD_WELD_DATA : WORD ;
    RBT22_STANDARD_WELD_DATA : WORD ;
    RBT23_STANDARD_WELD_DAT : WORD ;
    RBT24_STANDARD_WELD_DAT : WORD ;
    CHK_WORD : WORD ;
    TEST_TEMP : ARRAY  [1 .. 40 ] OF BYTE ;
   END_STRUCT ;
   S702_BT_CODE_2030 : STRUCT
    STATION_MAIN : WORD ;
    DISTINCTION_LH_RH : WORD ;
    STAION_NUMBER : WORD ;
    BODY_TYPE_1ST : WORD ;
    BODY_TYPE_OPTION : WORD ;
    RBT1_STANDARD_WELD_DATA : WORD ;
    RBT2_STANDARD_WELD_DATA : WORD ;
    RBT3_STANDARD_WELD_DATA : WORD ;
    RBT4_STANDARD_WELD_DATA : WORD ;
    RBT5_STANDARD_WELD_DATA : WORD ;
    RBT6_STANDARD_WELD_DATA : WORD ;
    RBT7_STANDARD_WELD_DATA : WORD ;
    RBT8_STANDARD_WELD_DATA : WORD ;
    RBT9_STANDARD_WELD_DATA : WORD ;
    RBT10_STANDARD_WELD_DATA : WORD ;
    RBT11_STANDARD_WELD_DATA : WORD ;
    RBT12_STANDARD_WELD_DATA : WORD ;
    RBT13_STANDARD_WELD_DATA : WORD ;
    RBT14_STANDARD_WELD_DATA : WORD ;
    RBT15_STANDARD_WELD_DATA : WORD ;
    RBT16_STANDARD_WELD_DATA : WORD ;
    RBT17_STANDARD_WELD_DATA : WORD ;
    RBT18_STANDARD_WELD_DATA : WORD ;
    RBT19_STANDARD_WELD_DATA : WORD ;
    RBT20_STANDARD_WELD_DATA : WORD ;
    RBT21_STANDARD_WELD_DATA : WORD ;
    RBT22_STANDARD_WELD_DATA : WORD ;
    RBT23_STANDARD_WELD_DAT : WORD ;
    RBT24_STANDARD_WELD_DAT : WORD ;
    CHK_WORD : WORD ;
    TEST_TEMP : ARRAY  [1 .. 40 ] OF BYTE ;
   END_STRUCT ;
   S704_BT_CODE_2011 : STRUCT
    STATION_MAIN : WORD ;
    DISTINCTION_LH_RH : WORD ;
    STAION_NUMBER : WORD ;
    BODY_TYPE_1ST : WORD ;
    BODY_TYPE_OPTION : WORD ;
    RBT1_STANDARD_WELD_DATA : WORD ;
    RBT2_STANDARD_WELD_DATA : WORD ;
    RBT3_STANDARD_WELD_DATA : WORD ;
    RBT4_STANDARD_WELD_DATA : WORD ;
    RBT5_STANDARD_WELD_DATA : WORD ;
    RBT6_STANDARD_WELD_DATA : WORD ;
    RBT7_STANDARD_WELD_DATA : WORD ;
    RBT8_STANDARD_WELD_DATA : WORD ;
    RBT9_STANDARD_WELD_DATA : WORD ;
    RBT10_STANDARD_WELD_DATA : WORD ;
    RBT11_STANDARD_WELD_DATA : WORD ;
    RBT12_STANDARD_WELD_DATA : WORD ;
    RBT13_STANDARD_WELD_DATA : WORD ;
    RBT14_STANDARD_WELD_DATA : WORD ;
    RBT15_STANDARD_WELD_DATA : WORD ;
    RBT16_STANDARD_WELD_DATA : WORD ;
    RBT17_STANDARD_WELD_DATA : WORD ;
    RBT18_STANDARD_WELD_DATA : WORD ;
    RBT19_STANDARD_WELD_DATA : WORD ;
    RBT20_STANDARD_WELD_DATA : WORD ;
    RBT21_STANDARD_WELD_DATA : WORD ;
    RBT22_STANDARD_WELD_DATA : WORD ;
    RBT23_STANDARD_WELD_DAT : WORD ;
    RBT24_STANDARD_WELD_DAT : WORD ;
    CHK_WORD : WORD ;
    TEST_TEMP : ARRAY  [1 .. 40 ] OF BYTE ;
   END_STRUCT ;
   S704_BT_CODE_2012 : STRUCT
    STATION_MAIN : WORD ;
    DISTINCTION_LH_RH : WORD ;
    STAION_NUMBER : WORD ;
    BODY_TYPE_1ST : WORD ;
    BODY_TYPE_OPTION : WORD ;
    RBT1_STANDARD_WELD_DATA : WORD ;
    RBT2_STANDARD_WELD_DATA : WORD ;
    RBT3_STANDARD_WELD_DATA : WORD ;
    RBT4_STANDARD_WELD_DATA : WORD ;
    RBT5_STANDARD_WELD_DATA : WORD ;
    RBT6_STANDARD_WELD_DATA : WORD ;
    RBT7_STANDARD_WELD_DATA : WORD ;
    RBT8_STANDARD_WELD_DATA : WORD ;
    RBT9_STANDARD_WELD_DATA : WORD ;
    RBT10_STANDARD_WELD_DATA : WORD ;
    RBT11_STANDARD_WELD_DATA : WORD ;
    RBT12_STANDARD_WELD_DATA : WORD ;
    RBT13_STANDARD_WELD_DATA : WORD ;
    RBT14_STANDARD_WELD_DATA : WORD ;
    RBT15_STANDARD_WELD_DATA : WORD ;
    RBT16_STANDARD_WELD_DATA : WORD ;
    RBT17_STANDARD_WELD_DATA : WORD ;
    RBT18_STANDARD_WELD_DATA : WORD ;
    RBT19_STANDARD_WELD_DATA : WORD ;
    RBT20_STANDARD_WELD_DATA : WORD ;
    RBT21_STANDARD_WELD_DATA : WORD ;
    RBT22_STANDARD_WELD_DATA : WORD ;
    RBT23_STANDARD_WELD_DAT : WORD ;
    RBT24_STANDARD_WELD_DAT : WORD ;
    CHK_WORD : WORD ;
    TEST_TEMP : ARRAY  [1 .. 40 ] OF BYTE ;
   END_STRUCT ;
   S704_BT_CODE_2013 : STRUCT
    STATION_MAIN : WORD ;
    DISTINCTION_LH_RH : WORD ;
    STAION_NUMBER : WORD ;
    BODY_TYPE_1ST : WORD ;
    BODY_TYPE_OPTION : WORD ;
    RBT1_STANDARD_WELD_DATA : WORD ;
    RBT2_STANDARD_WELD_DATA : WORD ;
    RBT3_STANDARD_WELD_DATA : WORD ;
    RBT4_STANDARD_WELD_DATA : WORD ;
    RBT5_STANDARD_WELD_DATA : WORD ;
    RBT6_STANDARD_WELD_DATA : WORD ;
    RBT7_STANDARD_WELD_DATA : WORD ;
    RBT8_STANDARD_WELD_DATA : WORD ;
    RBT9_STANDARD_WELD_DATA : WORD ;
    RBT10_STANDARD_WELD_DATA : WORD ;
    RBT11_STANDARD_WELD_DATA : WORD ;
    RBT12_STANDARD_WELD_DATA : WORD ;
    RBT13_STANDARD_WELD_DATA : WORD ;
    RBT14_STANDARD_WELD_DATA : WORD ;
    RBT15_STANDARD_WELD_DATA : WORD ;
    RBT16_STANDARD_WELD_DATA : WORD ;
    RBT17_STANDARD_WELD_DATA : WORD ;
    RBT18_STANDARD_WELD_DATA : WORD ;
    RBT19_STANDARD_WELD_DATA : WORD ;
    RBT20_STANDARD_WELD_DATA : WORD ;
    RBT21_STANDARD_WELD_DATA : WORD ;
    RBT22_STANDARD_WELD_DATA : WORD ;
    RBT23_STANDARD_WELD_DAT : WORD ;
    RBT24_STANDARD_WELD_DAT : WORD ;
    CHK_WORD : WORD ;
    TEST_TEMP : ARRAY  [1 .. 40 ] OF BYTE ;
   END_STRUCT ;
   S704_BT_CODE_2014 : STRUCT
    STATION_MAIN : WORD ;
    DISTINCTION_LH_RH : WORD ;
    STAION_NUMBER : WORD ;
    BODY_TYPE_1ST : WORD ;
    BODY_TYPE_OPTION : WORD ;
    RBT1_STANDARD_WELD_DATA : WORD ;
    RBT2_STANDARD_WELD_DATA : WORD ;
    RBT3_STANDARD_WELD_DATA : WORD ;
    RBT4_STANDARD_WELD_DATA : WORD ;
    RBT5_STANDARD_WELD_DATA : WORD ;
    RBT6_STANDARD_WELD_DATA : WORD ;
    RBT7_STANDARD_WELD_DATA : WORD ;
    RBT8_STANDARD_WELD_DATA : WORD ;
    RBT9_STANDARD_WELD_DATA : WORD ;
    RBT10_STANDARD_WELD_DATA : WORD ;
    RBT11_STANDARD_WELD_DATA : WORD ;
    RBT12_STANDARD_WELD_DATA : WORD ;
    RBT13_STANDARD_WELD_DATA : WORD ;
    RBT14_STANDARD_WELD_DATA : WORD ;
    RBT15_STANDARD_WELD_DATA : WORD ;
    RBT16_STANDARD_WELD_DATA : WORD ;
    RBT17_STANDARD_WELD_DATA : WORD ;
    RBT18_STANDARD_WELD_DATA : WORD ;
    RBT19_STANDARD_WELD_DATA : WORD ;
    RBT20_STANDARD_WELD_DATA : WORD ;
    RBT21_STANDARD_WELD_DATA : WORD ;
    RBT22_STANDARD_WELD_DATA : WORD ;
    RBT23_STANDARD_WELD_DAT : WORD ;
    RBT24_STANDARD_WELD_DAT : WORD ;
    CHK_WORD : WORD ;
    TEST_TEMP : ARRAY  [1 .. 40 ] OF BYTE ;
   END_STRUCT ;
   S704_BT_CODE_2015 : STRUCT
    STATION_MAIN : WORD ;
    DISTINCTION_LH_RH : WORD ;
    STAION_NUMBER : WORD ;
    BODY_TYPE_1ST : WORD ;
    BODY_TYPE_OPTION : WORD ;
    RBT1_STANDARD_WELD_DATA : WORD ;
    RBT2_STANDARD_WELD_DATA : WORD ;
    RBT3_STANDARD_WELD_DATA : WORD ;
    RBT4_STANDARD_WELD_DATA : WORD ;
    RBT5_STANDARD_WELD_DATA : WORD ;
    RBT6_STANDARD_WELD_DATA : WORD ;
    RBT7_STANDARD_WELD_DATA : WORD ;
    RBT8_STANDARD_WELD_DATA : WORD ;
    RBT9_STANDARD_WELD_DATA : WORD ;
    RBT10_STANDARD_WELD_DATA : WORD ;
    RBT11_STANDARD_WELD_DATA : WORD ;
    RBT12_STANDARD_WELD_DATA : WORD ;
    RBT13_STANDARD_WELD_DATA : WORD ;
    RBT14_STANDARD_WELD_DATA : WORD ;
    RBT15_STANDARD_WELD_DATA : WORD ;
    RBT16_STANDARD_WELD_DATA : WORD ;
    RBT17_STANDARD_WELD_DATA : WORD ;
    RBT18_STANDARD_WELD_DATA : WORD ;
    RBT19_STANDARD_WELD_DATA : WORD ;
    RBT20_STANDARD_WELD_DATA : WORD ;
    RBT21_STANDARD_WELD_DATA : WORD ;
    RBT22_STANDARD_WELD_DATA : WORD ;
    RBT23_STANDARD_WELD_DAT : WORD ;
    RBT24_STANDARD_WELD_DAT : WORD ;
    CHK_WORD : WORD ;
    TEST_TEMP : ARRAY  [1 .. 40 ] OF BYTE ;
   END_STRUCT ;
   S704_BT_CODE_2016 : STRUCT
    STATION_MAIN : WORD ;
    DISTINCTION_LH_RH : WORD ;
    STAION_NUMBER : WORD ;
    BODY_TYPE_1ST : WORD ;
    BODY_TYPE_OPTION : WORD ;
    RBT1_STANDARD_WELD_DATA : WORD ;
    RBT2_STANDARD_WELD_DATA : WORD ;
    RBT3_STANDARD_WELD_DATA : WORD ;
    RBT4_STANDARD_WELD_DATA : WORD ;
    RBT5_STANDARD_WELD_DATA : WORD ;
    RBT6_STANDARD_WELD_DATA : WORD ;
    RBT7_STANDARD_WELD_DATA : WORD ;
    RBT8_STANDARD_WELD_DATA : WORD ;
    RBT9_STANDARD_WELD_DATA : WORD ;
    RBT10_STANDARD_WELD_DATA : WORD ;
    RBT11_STANDARD_WELD_DATA : WORD ;
    RBT12_STANDARD_WELD_DATA : WORD ;
    RBT13_STANDARD_WELD_DATA : WORD ;
    RBT14_STANDARD_WELD_DATA : WORD ;
    RBT15_STANDARD_WELD_DATA : WORD ;
    RBT16_STANDARD_WELD_DATA : WORD ;
    RBT17_STANDARD_WELD_DATA : WORD ;
    RBT18_STANDARD_WELD_DATA : WORD ;
    RBT19_STANDARD_WELD_DATA : WORD ;
    RBT20_STANDARD_WELD_DATA : WORD ;
    RBT21_STANDARD_WELD_DATA : WORD ;
    RBT22_STANDARD_WELD_DATA : WORD ;
    RBT23_STANDARD_WELD_DAT : WORD ;
    RBT24_STANDARD_WELD_DAT : WORD ;
    CHK_WORD : WORD ;
    TEST_TEMP : ARRAY  [1 .. 40 ] OF BYTE ;
   END_STRUCT ;
   S704_BT_CODE_2017 : STRUCT
    STATION_MAIN : WORD ;
    DISTINCTION_LH_RH : WORD ;
    STAION_NUMBER : WORD ;
    BODY_TYPE_1ST : WORD ;
    BODY_TYPE_OPTION : WORD ;
    RBT1_STANDARD_WELD_DATA : WORD ;
    RBT2_STANDARD_WELD_DATA : WORD ;
    RBT3_STANDARD_WELD_DATA : WORD ;
    RBT4_STANDARD_WELD_DATA : WORD ;
    RBT5_STANDARD_WELD_DATA : WORD ;
    RBT6_STANDARD_WELD_DATA : WORD ;
    RBT7_STANDARD_WELD_DATA : WORD ;
    RBT8_STANDARD_WELD_DATA : WORD ;
    RBT9_STANDARD_WELD_DATA : WORD ;
    RBT10_STANDARD_WELD_DATA : WORD ;
    RBT11_STANDARD_WELD_DATA : WORD ;
    RBT12_STANDARD_WELD_DATA : WORD ;
    RBT13_STANDARD_WELD_DATA : WORD ;
    RBT14_STANDARD_WELD_DATA : WORD ;
    RBT15_STANDARD_WELD_DATA : WORD ;
    RBT16_STANDARD_WELD_DATA : WORD ;
    RBT17_STANDARD_WELD_DATA : WORD ;
    RBT18_STANDARD_WELD_DATA : WORD ;
    RBT19_STANDARD_WELD_DATA : WORD ;
    RBT20_STANDARD_WELD_DATA : WORD ;
    RBT21_STANDARD_WELD_DATA : WORD ;
    RBT22_STANDARD_WELD_DATA : WORD ;
    RBT23_STANDARD_WELD_DAT : WORD ;
    RBT24_STANDARD_WELD_DAT : WORD ;
    CHK_WORD : WORD ;
    TEST_TEMP : ARRAY  [1 .. 40 ] OF BYTE ;
   END_STRUCT ;
   S704_BT_CODE_2018 : STRUCT
    STATION_MAIN : WORD ;
    DISTINCTION_LH_RH : WORD ;
    STAION_NUMBER : WORD ;
    BODY_TYPE_1ST : WORD ;
    BODY_TYPE_OPTION : WORD ;
    RBT1_STANDARD_WELD_DATA : WORD ;
    RBT2_STANDARD_WELD_DATA : WORD ;
    RBT3_STANDARD_WELD_DATA : WORD ;
    RBT4_STANDARD_WELD_DATA : WORD ;
    RBT5_STANDARD_WELD_DATA : WORD ;
    RBT6_STANDARD_WELD_DATA : WORD ;
    RBT7_STANDARD_WELD_DATA : WORD ;
    RBT8_STANDARD_WELD_DATA : WORD ;
    RBT9_STANDARD_WELD_DATA : WORD ;
    RBT10_STANDARD_WELD_DATA : WORD ;
    RBT11_STANDARD_WELD_DATA : WORD ;
    RBT12_STANDARD_WELD_DATA : WORD ;
    RBT13_STANDARD_WELD_DATA : WORD ;
    RBT14_STANDARD_WELD_DATA : WORD ;
    RBT15_STANDARD_WELD_DATA : WORD ;
    RBT16_STANDARD_WELD_DATA : WORD ;
    RBT17_STANDARD_WELD_DATA : WORD ;
    RBT18_STANDARD_WELD_DATA : WORD ;
    RBT19_STANDARD_WELD_DATA : WORD ;
    RBT20_STANDARD_WELD_DATA : WORD ;
    RBT21_STANDARD_WELD_DATA : WORD ;
    RBT22_STANDARD_WELD_DATA : WORD ;
    RBT23_STANDARD_WELD_DAT : WORD ;
    RBT24_STANDARD_WELD_DAT : WORD ;
    CHK_WORD : WORD ;
    TEST_TEMP : ARRAY  [1 .. 40 ] OF BYTE ;
   END_STRUCT ;
   S704_BT_CODE_2019 : STRUCT
    STATION_MAIN : WORD ;
    DISTINCTION_LH_RH : WORD ;
    STAION_NUMBER : WORD ;
    BODY_TYPE_1ST : WORD ;
    BODY_TYPE_OPTION : WORD ;
    RBT1_STANDARD_WELD_DATA : WORD ;
    RBT2_STANDARD_WELD_DATA : WORD ;
    RBT3_STANDARD_WELD_DATA : WORD ;
    RBT4_STANDARD_WELD_DATA : WORD ;
    RBT5_STANDARD_WELD_DATA : WORD ;
    RBT6_STANDARD_WELD_DATA : WORD ;
    RBT7_STANDARD_WELD_DATA : WORD ;
    RBT8_STANDARD_WELD_DATA : WORD ;
    RBT9_STANDARD_WELD_DATA : WORD ;
    RBT10_STANDARD_WELD_DATA : WORD ;
    RBT11_STANDARD_WELD_DATA : WORD ;
    RBT12_STANDARD_WELD_DATA : WORD ;
    RBT13_STANDARD_WELD_DATA : WORD ;
    RBT14_STANDARD_WELD_DATA : WORD ;
    RBT15_STANDARD_WELD_DATA : WORD ;
    RBT16_STANDARD_WELD_DATA : WORD ;
    RBT17_STANDARD_WELD_DATA : WORD ;
    RBT18_STANDARD_WELD_DATA : WORD ;
    RBT19_STANDARD_WELD_DATA : WORD ;
    RBT20_STANDARD_WELD_DATA : WORD ;
    RBT21_STANDARD_WELD_DATA : WORD ;
    RBT22_STANDARD_WELD_DATA : WORD ;
    RBT23_STANDARD_WELD_DAT : WORD ;
    RBT24_STANDARD_WELD_DAT : WORD ;
    CHK_WORD : WORD ;
    TEST_TEMP : ARRAY  [1 .. 40 ] OF BYTE ;
   END_STRUCT ;
   S704_BT_CODE_2020 : STRUCT
    STATION_MAIN : WORD ;
    DISTINCTION_LH_RH : WORD ;
    STAION_NUMBER : WORD ;
    BODY_TYPE_1ST : WORD ;
    BODY_TYPE_OPTION : WORD ;
    RBT1_STANDARD_WELD_DATA : WORD ;
    RBT2_STANDARD_WELD_DATA : WORD ;
    RBT3_STANDARD_WELD_DATA : WORD ;
    RBT4_STANDARD_WELD_DATA : WORD ;
    RBT5_STANDARD_WELD_DATA : WORD ;
    RBT6_STANDARD_WELD_DATA : WORD ;
    RBT7_STANDARD_WELD_DATA : WORD ;
    RBT8_STANDARD_WELD_DATA : WORD ;
    RBT9_STANDARD_WELD_DATA : WORD ;
    RBT10_STANDARD_WELD_DATA : WORD ;
    RBT11_STANDARD_WELD_DATA : WORD ;
    RBT12_STANDARD_WELD_DATA : WORD ;
    RBT13_STANDARD_WELD_DATA : WORD ;
    RBT14_STANDARD_WELD_DATA : WORD ;
    RBT15_STANDARD_WELD_DATA : WORD ;
    RBT16_STANDARD_WELD_DATA : WORD ;
    RBT17_STANDARD_WELD_DATA : WORD ;
    RBT18_STANDARD_WELD_DATA : WORD ;
    RBT19_STANDARD_WELD_DATA : WORD ;
    RBT20_STANDARD_WELD_DATA : WORD ;
    RBT21_STANDARD_WELD_DATA : WORD ;
    RBT22_STANDARD_WELD_DATA : WORD ;
    RBT23_STANDARD_WELD_DAT : WORD ;
    RBT24_STANDARD_WELD_DAT : WORD ;
    CHK_WORD : WORD ;
    TEST_TEMP : ARRAY  [1 .. 40 ] OF BYTE ;
   END_STRUCT ;
   S704_BT_CODE_2021 : STRUCT
    STATION_MAIN : WORD ;
    DISTINCTION_LH_RH : WORD ;
    STAION_NUMBER : WORD ;
    BODY_TYPE_1ST : WORD ;
    BODY_TYPE_OPTION : WORD ;
    RBT1_STANDARD_WELD_DATA : WORD ;
    RBT2_STANDARD_WELD_DATA : WORD ;
    RBT3_STANDARD_WELD_DATA : WORD ;
    RBT4_STANDARD_WELD_DATA : WORD ;
    RBT5_STANDARD_WELD_DATA : WORD ;
    RBT6_STANDARD_WELD_DATA : WORD ;
    RBT7_STANDARD_WELD_DATA : WORD ;
    RBT8_STANDARD_WELD_DATA : WORD ;
    RBT9_STANDARD_WELD_DATA : WORD ;
    RBT10_STANDARD_WELD_DATA : WORD ;
    RBT11_STANDARD_WELD_DATA : WORD ;
    RBT12_STANDARD_WELD_DATA : WORD ;
    RBT13_STANDARD_WELD_DATA : WORD ;
    RBT14_STANDARD_WELD_DATA : WORD ;
    RBT15_STANDARD_WELD_DATA : WORD ;
    RBT16_STANDARD_WELD_DATA : WORD ;
    RBT17_STANDARD_WELD_DATA : WORD ;
    RBT18_STANDARD_WELD_DATA : WORD ;
    RBT19_STANDARD_WELD_DATA : WORD ;
    RBT20_STANDARD_WELD_DATA : WORD ;
    RBT21_STANDARD_WELD_DATA : WORD ;
    RBT22_STANDARD_WELD_DATA : WORD ;
    RBT23_STANDARD_WELD_DAT : WORD ;
    RBT24_STANDARD_WELD_DAT : WORD ;
    CHK_WORD : WORD ;
    TEST_TEMP : ARRAY  [1 .. 40 ] OF BYTE ;
   END_STRUCT ;
   S704_BT_CODE_2022 : STRUCT
    STATION_MAIN : WORD ;
    DISTINCTION_LH_RH : WORD ;
    STAION_NUMBER : WORD ;
    BODY_TYPE_1ST : WORD ;
    BODY_TYPE_OPTION : WORD ;
    RBT1_STANDARD_WELD_DATA : WORD ;
    RBT2_STANDARD_WELD_DATA : WORD ;
    RBT3_STANDARD_WELD_DATA : WORD ;
    RBT4_STANDARD_WELD_DATA : WORD ;
    RBT5_STANDARD_WELD_DATA : WORD ;
    RBT6_STANDARD_WELD_DATA : WORD ;
    RBT7_STANDARD_WELD_DATA : WORD ;
    RBT8_STANDARD_WELD_DATA : WORD ;
    RBT9_STANDARD_WELD_DATA : WORD ;
    RBT10_STANDARD_WELD_DATA : WORD ;
    RBT11_STANDARD_WELD_DATA : WORD ;
    RBT12_STANDARD_WELD_DATA : WORD ;
    RBT13_STANDARD_WELD_DATA : WORD ;
    RBT14_STANDARD_WELD_DATA : WORD ;
    RBT15_STANDARD_WELD_DATA : WORD ;
    RBT16_STANDARD_WELD_DATA : WORD ;
    RBT17_STANDARD_WELD_DATA : WORD ;
    RBT18_STANDARD_WELD_DATA : WORD ;
    RBT19_STANDARD_WELD_DATA : WORD ;
    RBT20_STANDARD_WELD_DATA : WORD ;
    RBT21_STANDARD_WELD_DATA : WORD ;
    RBT22_STANDARD_WELD_DATA : WORD ;
    RBT23_STANDARD_WELD_DAT : WORD ;
    RBT24_STANDARD_WELD_DAT : WORD ;
    CHK_WORD : WORD ;
    TEST_TEMP : ARRAY  [1 .. 40 ] OF BYTE ;
   END_STRUCT ;
   S704_BT_CODE_2023 : STRUCT
    STATION_MAIN : WORD ;
    DISTINCTION_LH_RH : WORD ;
    STAION_NUMBER : WORD ;
    BODY_TYPE_1ST : WORD ;
    BODY_TYPE_OPTION : WORD ;
    RBT1_STANDARD_WELD_DATA : WORD ;
    RBT2_STANDARD_WELD_DATA : WORD ;
    RBT3_STANDARD_WELD_DATA : WORD ;
    RBT4_STANDARD_WELD_DATA : WORD ;
    RBT5_STANDARD_WELD_DATA : WORD ;
    RBT6_STANDARD_WELD_DATA : WORD ;
    RBT7_STANDARD_WELD_DATA : WORD ;
    RBT8_STANDARD_WELD_DATA : WORD ;
    RBT9_STANDARD_WELD_DATA : WORD ;
    RBT10_STANDARD_WELD_DATA : WORD ;
    RBT11_STANDARD_WELD_DATA : WORD ;
    RBT12_STANDARD_WELD_DATA : WORD ;
    RBT13_STANDARD_WELD_DATA : WORD ;
    RBT14_STANDARD_WELD_DATA : WORD ;
    RBT15_STANDARD_WELD_DATA : WORD ;
    RBT16_STANDARD_WELD_DATA : WORD ;
    RBT17_STANDARD_WELD_DATA : WORD ;
    RBT18_STANDARD_WELD_DATA : WORD ;
    RBT19_STANDARD_WELD_DATA : WORD ;
    RBT20_STANDARD_WELD_DATA : WORD ;
    RBT21_STANDARD_WELD_DATA : WORD ;
    RBT22_STANDARD_WELD_DATA : WORD ;
    RBT23_STANDARD_WELD_DAT : WORD ;
    RBT24_STANDARD_WELD_DAT : WORD ;
    CHK_WORD : WORD ;
    TEST_TEMP : ARRAY  [1 .. 40 ] OF BYTE ;
   END_STRUCT ;
   S704_BT_CODE_2024 : STRUCT
    STATION_MAIN : WORD ;
    DISTINCTION_LH_RH : WORD ;
    STAION_NUMBER : WORD ;
    BODY_TYPE_1ST : WORD ;
    BODY_TYPE_OPTION : WORD ;
    RBT1_STANDARD_WELD_DATA : WORD ;
    RBT2_STANDARD_WELD_DATA : WORD ;
    RBT3_STANDARD_WELD_DATA : WORD ;
    RBT4_STANDARD_WELD_DATA : WORD ;
    RBT5_STANDARD_WELD_DATA : WORD ;
    RBT6_STANDARD_WELD_DATA : WORD ;
    RBT7_STANDARD_WELD_DATA : WORD ;
    RBT8_STANDARD_WELD_DATA : WORD ;
    RBT9_STANDARD_WELD_DATA : WORD ;
    RBT10_STANDARD_WELD_DATA : WORD ;
    RBT11_STANDARD_WELD_DATA : WORD ;
    RBT12_STANDARD_WELD_DATA : WORD ;
    RBT13_STANDARD_WELD_DATA : WORD ;
    RBT14_STANDARD_WELD_DATA : WORD ;
    RBT15_STANDARD_WELD_DATA : WORD ;
    RBT16_STANDARD_WELD_DATA : WORD ;
    RBT17_STANDARD_WELD_DATA : WORD ;
    RBT18_STANDARD_WELD_DATA : WORD ;
    RBT19_STANDARD_WELD_DATA : WORD ;
    RBT20_STANDARD_WELD_DATA : WORD ;
    RBT21_STANDARD_WELD_DATA : WORD ;
    RBT22_STANDARD_WELD_DATA : WORD ;
    RBT23_STANDARD_WELD_DAT : WORD ;
    RBT24_STANDARD_WELD_DAT : WORD ;
    CHK_WORD : WORD ;
    TEST_TEMP : ARRAY  [1 .. 40 ] OF BYTE ;
   END_STRUCT ;
   S704_BT_CODE_2025 : STRUCT
    STATION_MAIN : WORD ;
    DISTINCTION_LH_RH : WORD ;
    STAION_NUMBER : WORD ;
    BODY_TYPE_1ST : WORD ;
    BODY_TYPE_OPTION : WORD ;
    RBT1_STANDARD_WELD_DATA : WORD ;
    RBT2_STANDARD_WELD_DATA : WORD ;
    RBT3_STANDARD_WELD_DATA : WORD ;
    RBT4_STANDARD_WELD_DATA : WORD ;
    RBT5_STANDARD_WELD_DATA : WORD ;
    RBT6_STANDARD_WELD_DATA : WORD ;
    RBT7_STANDARD_WELD_DATA : WORD ;
    RBT8_STANDARD_WELD_DATA : WORD ;
    RBT9_STANDARD_WELD_DATA : WORD ;
    RBT10_STANDARD_WELD_DATA : WORD ;
    RBT11_STANDARD_WELD_DATA : WORD ;
    RBT12_STANDARD_WELD_DATA : WORD ;
    RBT13_STANDARD_WELD_DATA : WORD ;
    RBT14_STANDARD_WELD_DATA : WORD ;
    RBT15_STANDARD_WELD_DATA : WORD ;
    RBT16_STANDARD_WELD_DATA : WORD ;
    RBT17_STANDARD_WELD_DATA : WORD ;
    RBT18_STANDARD_WELD_DATA : WORD ;
    RBT19_STANDARD_WELD_DATA : WORD ;
    RBT20_STANDARD_WELD_DATA : WORD ;
    RBT21_STANDARD_WELD_DATA : WORD ;
    RBT22_STANDARD_WELD_DATA : WORD ;
    RBT23_STANDARD_WELD_DAT : WORD ;
    RBT24_STANDARD_WELD_DAT : WORD ;
    CHK_WORD : WORD ;
    TEST_TEMP : ARRAY  [1 .. 40 ] OF BYTE ;
   END_STRUCT ;
   S704_BT_CODE_2026 : STRUCT
    STATION_MAIN : WORD ;
    DISTINCTION_LH_RH : WORD ;
    STAION_NUMBER : WORD ;
    BODY_TYPE_1ST : WORD ;
    BODY_TYPE_OPTION : WORD ;
    RBT1_STANDARD_WELD_DATA : WORD ;
    RBT2_STANDARD_WELD_DATA : WORD ;
    RBT3_STANDARD_WELD_DATA : WORD ;
    RBT4_STANDARD_WELD_DATA : WORD ;
    RBT5_STANDARD_WELD_DATA : WORD ;
    RBT6_STANDARD_WELD_DATA : WORD ;
    RBT7_STANDARD_WELD_DATA : WORD ;
    RBT8_STANDARD_WELD_DATA : WORD ;
    RBT9_STANDARD_WELD_DATA : WORD ;
    RBT10_STANDARD_WELD_DATA : WORD ;
    RBT11_STANDARD_WELD_DATA : WORD ;
    RBT12_STANDARD_WELD_DATA : WORD ;
    RBT13_STANDARD_WELD_DATA : WORD ;
    RBT14_STANDARD_WELD_DATA : WORD ;
    RBT15_STANDARD_WELD_DATA : WORD ;
    RBT16_STANDARD_WELD_DATA : WORD ;
    RBT17_STANDARD_WELD_DATA : WORD ;
    RBT18_STANDARD_WELD_DATA : WORD ;
    RBT19_STANDARD_WELD_DATA : WORD ;
    RBT20_STANDARD_WELD_DATA : WORD ;
    RBT21_STANDARD_WELD_DATA : WORD ;
    RBT22_STANDARD_WELD_DATA : WORD ;
    RBT23_STANDARD_WELD_DAT : WORD ;
    RBT24_STANDARD_WELD_DAT : WORD ;
    CHK_WORD : WORD ;
    TEST_TEMP : ARRAY  [1 .. 40 ] OF BYTE ;
   END_STRUCT ;
   S704_BT_CODE_2027 : STRUCT
    STATION_MAIN : WORD ;
    DISTINCTION_LH_RH : WORD ;
    STAION_NUMBER : WORD ;
    BODY_TYPE_1ST : WORD ;
    BODY_TYPE_OPTION : WORD ;
    RBT1_STANDARD_WELD_DATA : WORD ;
    RBT2_STANDARD_WELD_DATA : WORD ;
    RBT3_STANDARD_WELD_DATA : WORD ;
    RBT4_STANDARD_WELD_DATA : WORD ;
    RBT5_STANDARD_WELD_DATA : WORD ;
    RBT6_STANDARD_WELD_DATA : WORD ;
    RBT7_STANDARD_WELD_DATA : WORD ;
    RBT8_STANDARD_WELD_DATA : WORD ;
    RBT9_STANDARD_WELD_DATA : WORD ;
    RBT10_STANDARD_WELD_DATA : WORD ;
    RBT11_STANDARD_WELD_DATA : WORD ;
    RBT12_STANDARD_WELD_DATA : WORD ;
    RBT13_STANDARD_WELD_DATA : WORD ;
    RBT14_STANDARD_WELD_DATA : WORD ;
    RBT15_STANDARD_WELD_DATA : WORD ;
    RBT16_STANDARD_WELD_DATA : WORD ;
    RBT17_STANDARD_WELD_DATA : WORD ;
    RBT18_STANDARD_WELD_DATA : WORD ;
    RBT19_STANDARD_WELD_DATA : WORD ;
    RBT20_STANDARD_WELD_DATA : WORD ;
    RBT21_STANDARD_WELD_DATA : WORD ;
    RBT22_STANDARD_WELD_DATA : WORD ;
    RBT23_STANDARD_WELD_DAT : WORD ;
    RBT24_STANDARD_WELD_DAT : WORD ;
    CHK_WORD : WORD ;
    TEST_TEMP : ARRAY  [1 .. 40 ] OF BYTE ;
   END_STRUCT ;
   S704_BT_CODE_2028 : STRUCT
    STATION_MAIN : WORD ;
    DISTINCTION_LH_RH : WORD ;
    STAION_NUMBER : WORD ;
    BODY_TYPE_1ST : WORD ;
    BODY_TYPE_OPTION : WORD ;
    RBT1_STANDARD_WELD_DATA : WORD ;
    RBT2_STANDARD_WELD_DATA : WORD ;
    RBT3_STANDARD_WELD_DATA : WORD ;
    RBT4_STANDARD_WELD_DATA : WORD ;
    RBT5_STANDARD_WELD_DATA : WORD ;
    RBT6_STANDARD_WELD_DATA : WORD ;
    RBT7_STANDARD_WELD_DATA : WORD ;
    RBT8_STANDARD_WELD_DATA : WORD ;
    RBT9_STANDARD_WELD_DATA : WORD ;
    RBT10_STANDARD_WELD_DATA : WORD ;
    RBT11_STANDARD_WELD_DATA : WORD ;
    RBT12_STANDARD_WELD_DATA : WORD ;
    RBT13_STANDARD_WELD_DATA : WORD ;
    RBT14_STANDARD_WELD_DATA : WORD ;
    RBT15_STANDARD_WELD_DATA : WORD ;
    RBT16_STANDARD_WELD_DATA : WORD ;
    RBT17_STANDARD_WELD_DATA : WORD ;
    RBT18_STANDARD_WELD_DATA : WORD ;
    RBT19_STANDARD_WELD_DATA : WORD ;
    RBT20_STANDARD_WELD_DATA : WORD ;
    RBT21_STANDARD_WELD_DATA : WORD ;
    RBT22_STANDARD_WELD_DATA : WORD ;
    RBT23_STANDARD_WELD_DAT : WORD ;
    RBT24_STANDARD_WELD_DAT : WORD ;
    CHK_WORD : WORD ;
    TEST_TEMP : ARRAY  [1 .. 40 ] OF BYTE ;
   END_STRUCT ;
   S704_BT_CODE_2029 : STRUCT
    STATION_MAIN : WORD ;
    DISTINCTION_LH_RH : WORD ;
    STAION_NUMBER : WORD ;
    BODY_TYPE_1ST : WORD ;
    BODY_TYPE_OPTION : WORD ;
    RBT1_STANDARD_WELD_DATA : WORD ;
    RBT2_STANDARD_WELD_DATA : WORD ;
    RBT3_STANDARD_WELD_DATA : WORD ;
    RBT4_STANDARD_WELD_DATA : WORD ;
    RBT5_STANDARD_WELD_DATA : WORD ;
    RBT6_STANDARD_WELD_DATA : WORD ;
    RBT7_STANDARD_WELD_DATA : WORD ;
    RBT8_STANDARD_WELD_DATA : WORD ;
    RBT9_STANDARD_WELD_DATA : WORD ;
    RBT10_STANDARD_WELD_DATA : WORD ;
    RBT11_STANDARD_WELD_DATA : WORD ;
    RBT12_STANDARD_WELD_DATA : WORD ;
    RBT13_STANDARD_WELD_DATA : WORD ;
    RBT14_STANDARD_WELD_DATA : WORD ;
    RBT15_STANDARD_WELD_DATA : WORD ;
    RBT16_STANDARD_WELD_DATA : WORD ;
    RBT17_STANDARD_WELD_DATA : WORD ;
    RBT18_STANDARD_WELD_DATA : WORD ;
    RBT19_STANDARD_WELD_DATA : WORD ;
    RBT20_STANDARD_WELD_DATA : WORD ;
    RBT21_STANDARD_WELD_DATA : WORD ;
    RBT22_STANDARD_WELD_DATA : WORD ;
    RBT23_STANDARD_WELD_DAT : WORD ;
    RBT24_STANDARD_WELD_DAT : WORD ;
    CHK_WORD : WORD ;
    TEST_TEMP : ARRAY  [1 .. 40 ] OF BYTE ;
   END_STRUCT ;
   S704_BT_CODE_2030 : STRUCT
    STATION_MAIN : WORD ;
    DISTINCTION_LH_RH : WORD ;
    STAION_NUMBER : WORD ;
    BODY_TYPE_1ST : WORD ;
    BODY_TYPE_OPTION : WORD ;
    RBT1_STANDARD_WELD_DATA : WORD ;
    RBT2_STANDARD_WELD_DATA : WORD ;
    RBT3_STANDARD_WELD_DATA : WORD ;
    RBT4_STANDARD_WELD_DATA : WORD ;
    RBT5_STANDARD_WELD_DATA : WORD ;
    RBT6_STANDARD_WELD_DATA : WORD ;
    RBT7_STANDARD_WELD_DATA : WORD ;
    RBT8_STANDARD_WELD_DATA : WORD ;
    RBT9_STANDARD_WELD_DATA : WORD ;
    RBT10_STANDARD_WELD_DATA : WORD ;
    RBT11_STANDARD_WELD_DATA : WORD ;
    RBT12_STANDARD_WELD_DATA : WORD ;
    RBT13_STANDARD_WELD_DATA : WORD ;
    RBT14_STANDARD_WELD_DATA : WORD ;
    RBT15_STANDARD_WELD_DATA : WORD ;
    RBT16_STANDARD_WELD_DATA : WORD ;
    RBT17_STANDARD_WELD_DATA : WORD ;
    RBT18_STANDARD_WELD_DATA : WORD ;
    RBT19_STANDARD_WELD_DATA : WORD ;
    RBT20_STANDARD_WELD_DATA : WORD ;
    RBT21_STANDARD_WELD_DATA : WORD ;
    RBT22_STANDARD_WELD_DATA : WORD ;
    RBT23_STANDARD_WELD_DAT : WORD ;
    RBT24_STANDARD_WELD_DAT : WORD ;
    CHK_WORD : WORD ;
    TEST_TEMP : ARRAY  [1 .. 40 ] OF BYTE ;
   END_STRUCT ;
   S702_BT_CODE_2101 : STRUCT
    STATION_MAIN : WORD ;
    DISTINCTION_LH_RH : WORD ;
    STAION_NUMBER : WORD ;
    BODY_TYPE_1ST : WORD ;
    BODY_TYPE_OPTION : WORD ;
    RBT1_STANDARD_WELD_DATA : WORD ;
    RBT2_STANDARD_WELD_DATA : WORD ;
    RBT3_STANDARD_WELD_DATA : WORD ;
    RBT4_STANDARD_WELD_DATA : WORD ;
    RBT5_STANDARD_WELD_DATA : WORD ;
    RBT6_STANDARD_WELD_DATA : WORD ;
    RBT7_STANDARD_WELD_DATA : WORD ;
    RBT8_STANDARD_WELD_DATA : WORD ;
    RBT9_STANDARD_WELD_DATA : WORD ;
    RBT10_STANDARD_WELD_DATA : WORD ;
    RBT11_STANDARD_WELD_DATA : WORD ;
    RBT12_STANDARD_WELD_DATA : WORD ;
    RBT13_STANDARD_WELD_DATA : WORD ;
    RBT14_STANDARD_WELD_DATA : WORD ;
    RBT15_STANDARD_WELD_DATA : WORD ;
    RBT16_STANDARD_WELD_DATA : WORD ;
    RBT17_STANDARD_WELD_DATA : WORD ;
    RBT18_STANDARD_WELD_DATA : WORD ;
    RBT19_STANDARD_WELD_DATA : WORD ;
    RBT20_STANDARD_WELD_DATA : WORD ;
    RBT21_STANDARD_WELD_DATA : WORD ;
    RBT22_STANDARD_WELD_DATA : WORD ;
    RBT23_STANDARD_WELD_DAT : WORD ;
    RBT24_STANDARD_WELD_DAT : WORD ;
    CHK_WORD : WORD ;
    TEST_TEMP : ARRAY  [1 .. 40 ] OF BYTE ;
   END_STRUCT ;
   S702_BT_CODE_2102 : STRUCT
    STATION_MAIN : WORD ;
    DISTINCTION_LH_RH : WORD ;
    STAION_NUMBER : WORD ;
    BODY_TYPE_1ST : WORD ;
    BODY_TYPE_OPTION : WORD ;
    RBT1_STANDARD_WELD_DATA : WORD ;
    RBT2_STANDARD_WELD_DATA : WORD ;
    RBT3_STANDARD_WELD_DATA : WORD ;
    RBT4_STANDARD_WELD_DATA : WORD ;
    RBT5_STANDARD_WELD_DATA : WORD ;
    RBT6_STANDARD_WELD_DATA : WORD ;
    RBT7_STANDARD_WELD_DATA : WORD ;
    RBT8_STANDARD_WELD_DATA : WORD ;
    RBT9_STANDARD_WELD_DATA : WORD ;
    RBT10_STANDARD_WELD_DATA : WORD ;
    RBT11_STANDARD_WELD_DATA : WORD ;
    RBT12_STANDARD_WELD_DATA : WORD ;
    RBT13_STANDARD_WELD_DATA : WORD ;
    RBT14_STANDARD_WELD_DATA : WORD ;
    RBT15_STANDARD_WELD_DATA : WORD ;
    RBT16_STANDARD_WELD_DATA : WORD ;
    RBT17_STANDARD_WELD_DATA : WORD ;
    RBT18_STANDARD_WELD_DATA : WORD ;
    RBT19_STANDARD_WELD_DATA : WORD ;
    RBT20_STANDARD_WELD_DATA : WORD ;
    RBT21_STANDARD_WELD_DATA : WORD ;
    RBT22_STANDARD_WELD_DATA : WORD ;
    RBT23_STANDARD_WELD_DAT : WORD ;
    RBT24_STANDARD_WELD_DAT : WORD ;
    CHK_WORD : WORD ;
    TEST_TEMP : ARRAY  [1 .. 40 ] OF BYTE ;
   END_STRUCT ;
   S702_BT_CODE_2103 : STRUCT
    STATION_MAIN : WORD ;
    DISTINCTION_LH_RH : WORD ;
    STAION_NUMBER : WORD ;
    BODY_TYPE_1ST : WORD ;
    BODY_TYPE_OPTION : WORD ;
    RBT1_STANDARD_WELD_DATA : WORD ;
    RBT2_STANDARD_WELD_DATA : WORD ;
    RBT3_STANDARD_WELD_DATA : WORD ;
    RBT4_STANDARD_WELD_DATA : WORD ;
    RBT5_STANDARD_WELD_DATA : WORD ;
    RBT6_STANDARD_WELD_DATA : WORD ;
    RBT7_STANDARD_WELD_DATA : WORD ;
    RBT8_STANDARD_WELD_DATA : WORD ;
    RBT9_STANDARD_WELD_DATA : WORD ;
    RBT10_STANDARD_WELD_DATA : WORD ;
    RBT11_STANDARD_WELD_DATA : WORD ;
    RBT12_STANDARD_WELD_DATA : WORD ;
    RBT13_STANDARD_WELD_DATA : WORD ;
    RBT14_STANDARD_WELD_DATA : WORD ;
    RBT15_STANDARD_WELD_DATA : WORD ;
    RBT16_STANDARD_WELD_DATA : WORD ;
    RBT17_STANDARD_WELD_DATA : WORD ;
    RBT18_STANDARD_WELD_DATA : WORD ;
    RBT19_STANDARD_WELD_DATA : WORD ;
    RBT20_STANDARD_WELD_DATA : WORD ;
    RBT21_STANDARD_WELD_DATA : WORD ;
    RBT22_STANDARD_WELD_DATA : WORD ;
    RBT23_STANDARD_WELD_DAT : WORD ;
    RBT24_STANDARD_WELD_DAT : WORD ;
    CHK_WORD : WORD ;
    TEST_TEMP : ARRAY  [1 .. 40 ] OF BYTE ;
   END_STRUCT ;
   S702_BT_CODE_2104 : STRUCT
    STATION_MAIN : WORD ;
    DISTINCTION_LH_RH : WORD ;
    STAION_NUMBER : WORD ;
    BODY_TYPE_1ST : WORD ;
    BODY_TYPE_OPTION : WORD ;
    RBT1_STANDARD_WELD_DATA : WORD ;
    RBT2_STANDARD_WELD_DATA : WORD ;
    RBT3_STANDARD_WELD_DATA : WORD ;
    RBT4_STANDARD_WELD_DATA : WORD ;
    RBT5_STANDARD_WELD_DATA : WORD ;
    RBT6_STANDARD_WELD_DATA : WORD ;
    RBT7_STANDARD_WELD_DATA : WORD ;
    RBT8_STANDARD_WELD_DATA : WORD ;
    RBT9_STANDARD_WELD_DATA : WORD ;
    RBT10_STANDARD_WELD_DATA : WORD ;
    RBT11_STANDARD_WELD_DATA : WORD ;
    RBT12_STANDARD_WELD_DATA : WORD ;
    RBT13_STANDARD_WELD_DATA : WORD ;
    RBT14_STANDARD_WELD_DATA : WORD ;
    RBT15_STANDARD_WELD_DATA : WORD ;
    RBT16_STANDARD_WELD_DATA : WORD ;
    RBT17_STANDARD_WELD_DATA : WORD ;
    RBT18_STANDARD_WELD_DATA : WORD ;
    RBT19_STANDARD_WELD_DATA : WORD ;
    RBT20_STANDARD_WELD_DATA : WORD ;
    RBT21_STANDARD_WELD_DATA : WORD ;
    RBT22_STANDARD_WELD_DATA : WORD ;
    RBT23_STANDARD_WELD_DAT : WORD ;
    RBT24_STANDARD_WELD_DAT : WORD ;
    CHK_WORD : WORD ;
    TEST_TEMP : ARRAY  [1 .. 40 ] OF BYTE ;
   END_STRUCT ;
   S702_BT_CODE_2105 : STRUCT
    STATION_MAIN : WORD ;
    DISTINCTION_LH_RH : WORD ;
    STAION_NUMBER : WORD ;
    BODY_TYPE_1ST : WORD ;
    BODY_TYPE_OPTION : WORD ;
    RBT1_STANDARD_WELD_DATA : WORD ;
    RBT2_STANDARD_WELD_DATA : WORD ;
    RBT3_STANDARD_WELD_DATA : WORD ;
    RBT4_STANDARD_WELD_DATA : WORD ;
    RBT5_STANDARD_WELD_DATA : WORD ;
    RBT6_STANDARD_WELD_DATA : WORD ;
    RBT7_STANDARD_WELD_DATA : WORD ;
    RBT8_STANDARD_WELD_DATA : WORD ;
    RBT9_STANDARD_WELD_DATA : WORD ;
    RBT10_STANDARD_WELD_DATA : WORD ;
    RBT11_STANDARD_WELD_DATA : WORD ;
    RBT12_STANDARD_WELD_DATA : WORD ;
    RBT13_STANDARD_WELD_DATA : WORD ;
    RBT14_STANDARD_WELD_DATA : WORD ;
    RBT15_STANDARD_WELD_DATA : WORD ;
    RBT16_STANDARD_WELD_DATA : WORD ;
    RBT17_STANDARD_WELD_DATA : WORD ;
    RBT18_STANDARD_WELD_DATA : WORD ;
    RBT19_STANDARD_WELD_DATA : WORD ;
    RBT20_STANDARD_WELD_DATA : WORD ;
    RBT21_STANDARD_WELD_DATA : WORD ;
    RBT22_STANDARD_WELD_DATA : WORD ;
    RBT23_STANDARD_WELD_DAT : WORD ;
    RBT24_STANDARD_WELD_DAT : WORD ;
    CHK_WORD : WORD ;
    TEST_TEMP : ARRAY  [1 .. 40 ] OF BYTE ;
   END_STRUCT ;
   S702_BT_CODE_2106 : STRUCT
    STATION_MAIN : WORD ;
    DISTINCTION_LH_RH : WORD ;
    STAION_NUMBER : WORD ;
    BODY_TYPE_1ST : WORD ;
    BODY_TYPE_OPTION : WORD ;
    RBT1_STANDARD_WELD_DATA : WORD ;
    RBT2_STANDARD_WELD_DATA : WORD ;
    RBT3_STANDARD_WELD_DATA : WORD ;
    RBT4_STANDARD_WELD_DATA : WORD ;
    RBT5_STANDARD_WELD_DATA : WORD ;
    RBT6_STANDARD_WELD_DATA : WORD ;
    RBT7_STANDARD_WELD_DATA : WORD ;
    RBT8_STANDARD_WELD_DATA : WORD ;
    RBT9_STANDARD_WELD_DATA : WORD ;
    RBT10_STANDARD_WELD_DATA : WORD ;
    RBT11_STANDARD_WELD_DATA : WORD ;
    RBT12_STANDARD_WELD_DATA : WORD ;
    RBT13_STANDARD_WELD_DATA : WORD ;
    RBT14_STANDARD_WELD_DATA : WORD ;
    RBT15_STANDARD_WELD_DATA : WORD ;
    RBT16_STANDARD_WELD_DATA : WORD ;
    RBT17_STANDARD_WELD_DATA : WORD ;
    RBT18_STANDARD_WELD_DATA : WORD ;
    RBT19_STANDARD_WELD_DATA : WORD ;
    RBT20_STANDARD_WELD_DATA : WORD ;
    RBT21_STANDARD_WELD_DATA : WORD ;
    RBT22_STANDARD_WELD_DATA : WORD ;
    RBT23_STANDARD_WELD_DAT : WORD ;
    RBT24_STANDARD_WELD_DAT : WORD ;
    CHK_WORD : WORD ;
    TEST_TEMP : ARRAY  [1 .. 40 ] OF BYTE ;
   END_STRUCT ;
   S702_BT_CODE_2107 : STRUCT
    STATION_MAIN : WORD ;
    DISTINCTION_LH_RH : WORD ;
    STAION_NUMBER : WORD ;
    BODY_TYPE_1ST : WORD ;
    BODY_TYPE_OPTION : WORD ;
    RBT1_STANDARD_WELD_DATA : WORD ;
    RBT2_STANDARD_WELD_DATA : WORD ;
    RBT3_STANDARD_WELD_DATA : WORD ;
    RBT4_STANDARD_WELD_DATA : WORD ;
    RBT5_STANDARD_WELD_DATA : WORD ;
    RBT6_STANDARD_WELD_DATA : WORD ;
    RBT7_STANDARD_WELD_DATA : WORD ;
    RBT8_STANDARD_WELD_DATA : WORD ;
    RBT9_STANDARD_WELD_DATA : WORD ;
    RBT10_STANDARD_WELD_DATA : WORD ;
    RBT11_STANDARD_WELD_DATA : WORD ;
    RBT12_STANDARD_WELD_DATA : WORD ;
    RBT13_STANDARD_WELD_DATA : WORD ;
    RBT14_STANDARD_WELD_DATA : WORD ;
    RBT15_STANDARD_WELD_DATA : WORD ;
    RBT16_STANDARD_WELD_DATA : WORD ;
    RBT17_STANDARD_WELD_DATA : WORD ;
    RBT18_STANDARD_WELD_DATA : WORD ;
    RBT19_STANDARD_WELD_DATA : WORD ;
    RBT20_STANDARD_WELD_DATA : WORD ;
    RBT21_STANDARD_WELD_DATA : WORD ;
    RBT22_STANDARD_WELD_DATA : WORD ;
    RBT23_STANDARD_WELD_DAT : WORD ;
    RBT24_STANDARD_WELD_DAT : WORD ;
    CHK_WORD : WORD ;
    TEST_TEMP : ARRAY  [1 .. 40 ] OF BYTE ;
   END_STRUCT ;
   S702_BT_CODE_2108 : STRUCT
    STATION_MAIN : WORD ;
    DISTINCTION_LH_RH : WORD ;
    STAION_NUMBER : WORD ;
    BODY_TYPE_1ST : WORD ;
    BODY_TYPE_OPTION : WORD ;
    RBT1_STANDARD_WELD_DATA : WORD ;
    RBT2_STANDARD_WELD_DATA : WORD ;
    RBT3_STANDARD_WELD_DATA : WORD ;
    RBT4_STANDARD_WELD_DATA : WORD ;
    RBT5_STANDARD_WELD_DATA : WORD ;
    RBT6_STANDARD_WELD_DATA : WORD ;
    RBT7_STANDARD_WELD_DATA : WORD ;
    RBT8_STANDARD_WELD_DATA : WORD ;
    RBT9_STANDARD_WELD_DATA : WORD ;
    RBT10_STANDARD_WELD_DATA : WORD ;
    RBT11_STANDARD_WELD_DATA : WORD ;
    RBT12_STANDARD_WELD_DATA : WORD ;
    RBT13_STANDARD_WELD_DATA : WORD ;
    RBT14_STANDARD_WELD_DATA : WORD ;
    RBT15_STANDARD_WELD_DATA : WORD ;
    RBT16_STANDARD_WELD_DATA : WORD ;
    RBT17_STANDARD_WELD_DATA : WORD ;
    RBT18_STANDARD_WELD_DATA : WORD ;
    RBT19_STANDARD_WELD_DATA : WORD ;
    RBT20_STANDARD_WELD_DATA : WORD ;
    RBT21_STANDARD_WELD_DATA : WORD ;
    RBT22_STANDARD_WELD_DATA : WORD ;
    RBT23_STANDARD_WELD_DAT : WORD ;
    RBT24_STANDARD_WELD_DAT : WORD ;
    CHK_WORD : WORD ;
    TEST_TEMP : ARRAY  [1 .. 40 ] OF BYTE ;
   END_STRUCT ;
   S702_BT_CODE_2109 : STRUCT
    STATION_MAIN : WORD ;
    DISTINCTION_LH_RH : WORD ;
    STAION_NUMBER : WORD ;
    BODY_TYPE_1ST : WORD ;
    BODY_TYPE_OPTION : WORD ;
    RBT1_STANDARD_WELD_DATA : WORD ;
    RBT2_STANDARD_WELD_DATA : WORD ;
    RBT3_STANDARD_WELD_DATA : WORD ;
    RBT4_STANDARD_WELD_DATA : WORD ;
    RBT5_STANDARD_WELD_DATA : WORD ;
    RBT6_STANDARD_WELD_DATA : WORD ;
    RBT7_STANDARD_WELD_DATA : WORD ;
    RBT8_STANDARD_WELD_DATA : WORD ;
    RBT9_STANDARD_WELD_DATA : WORD ;
    RBT10_STANDARD_WELD_DATA : WORD ;
    RBT11_STANDARD_WELD_DATA : WORD ;
    RBT12_STANDARD_WELD_DATA : WORD ;
    RBT13_STANDARD_WELD_DATA : WORD ;
    RBT14_STANDARD_WELD_DATA : WORD ;
    RBT15_STANDARD_WELD_DATA : WORD ;
    RBT16_STANDARD_WELD_DATA : WORD ;
    RBT17_STANDARD_WELD_DATA : WORD ;
    RBT18_STANDARD_WELD_DATA : WORD ;
    RBT19_STANDARD_WELD_DATA : WORD ;
    RBT20_STANDARD_WELD_DATA : WORD ;
    RBT21_STANDARD_WELD_DATA : WORD ;
    RBT22_STANDARD_WELD_DATA : WORD ;
    RBT23_STANDARD_WELD_DAT : WORD ;
    RBT24_STANDARD_WELD_DAT : WORD ;
    CHK_WORD : WORD ;
    TEST_TEMP : ARRAY  [1 .. 40 ] OF BYTE ;
   END_STRUCT ;
   S702_BT_CODE_2110 : STRUCT
    STATION_MAIN : WORD ;
    DISTINCTION_LH_RH : WORD ;
    STAION_NUMBER : WORD ;
    BODY_TYPE_1ST : WORD ;
    BODY_TYPE_OPTION : WORD ;
    RBT1_STANDARD_WELD_DATA : WORD ;
    RBT2_STANDARD_WELD_DATA : WORD ;
    RBT3_STANDARD_WELD_DATA : WORD ;
    RBT4_STANDARD_WELD_DATA : WORD ;
    RBT5_STANDARD_WELD_DATA : WORD ;
    RBT6_STANDARD_WELD_DATA : WORD ;
    RBT7_STANDARD_WELD_DATA : WORD ;
    RBT8_STANDARD_WELD_DATA : WORD ;
    RBT9_STANDARD_WELD_DATA : WORD ;
    RBT10_STANDARD_WELD_DATA : WORD ;
    RBT11_STANDARD_WELD_DATA : WORD ;
    RBT12_STANDARD_WELD_DATA : WORD ;
    RBT13_STANDARD_WELD_DATA : WORD ;
    RBT14_STANDARD_WELD_DATA : WORD ;
    RBT15_STANDARD_WELD_DATA : WORD ;
    RBT16_STANDARD_WELD_DATA : WORD ;
    RBT17_STANDARD_WELD_DATA : WORD ;
    RBT18_STANDARD_WELD_DATA : WORD ;
    RBT19_STANDARD_WELD_DATA : WORD ;
    RBT20_STANDARD_WELD_DATA : WORD ;
    RBT21_STANDARD_WELD_DATA : WORD ;
    RBT22_STANDARD_WELD_DATA : WORD ;
    RBT23_STANDARD_WELD_DAT : WORD ;
    RBT24_STANDARD_WELD_DAT : WORD ;
    CHK_WORD : WORD ;
    TEST_TEMP : ARRAY  [1 .. 40 ] OF BYTE ;
   END_STRUCT ;
   S702_BT_CODE_2111 : STRUCT
    STATION_MAIN : WORD ;
    DISTINCTION_LH_RH : WORD ;
    STAION_NUMBER : WORD ;
    BODY_TYPE_1ST : WORD ;
    BODY_TYPE_OPTION : WORD ;
    RBT1_STANDARD_WELD_DATA : WORD ;
    RBT2_STANDARD_WELD_DATA : WORD ;
    RBT3_STANDARD_WELD_DATA : WORD ;
    RBT4_STANDARD_WELD_DATA : WORD ;
    RBT5_STANDARD_WELD_DATA : WORD ;
    RBT6_STANDARD_WELD_DATA : WORD ;
    RBT7_STANDARD_WELD_DATA : WORD ;
    RBT8_STANDARD_WELD_DATA : WORD ;
    RBT9_STANDARD_WELD_DATA : WORD ;
    RBT10_STANDARD_WELD_DATA : WORD ;
    RBT11_STANDARD_WELD_DATA : WORD ;
    RBT12_STANDARD_WELD_DATA : WORD ;
    RBT13_STANDARD_WELD_DATA : WORD ;
    RBT14_STANDARD_WELD_DATA : WORD ;
    RBT15_STANDARD_WELD_DATA : WORD ;
    RBT16_STANDARD_WELD_DATA : WORD ;
    RBT17_STANDARD_WELD_DATA : WORD ;
    RBT18_STANDARD_WELD_DATA : WORD ;
    RBT19_STANDARD_WELD_DATA : WORD ;
    RBT20_STANDARD_WELD_DATA : WORD ;
    RBT21_STANDARD_WELD_DATA : WORD ;
    RBT22_STANDARD_WELD_DATA : WORD ;
    RBT23_STANDARD_WELD_DAT : WORD ;
    RBT24_STANDARD_WELD_DAT : WORD ;
    CHK_WORD : WORD ;
    TEST_TEMP : ARRAY  [1 .. 40 ] OF BYTE ;
   END_STRUCT ;
   S702_BT_CODE_2112 : STRUCT
    STATION_MAIN : WORD ;
    DISTINCTION_LH_RH : WORD ;
    STAION_NUMBER : WORD ;
    BODY_TYPE_1ST : WORD ;
    BODY_TYPE_OPTION : WORD ;
    RBT1_STANDARD_WELD_DATA : WORD ;
    RBT2_STANDARD_WELD_DATA : WORD ;
    RBT3_STANDARD_WELD_DATA : WORD ;
    RBT4_STANDARD_WELD_DATA : WORD ;
    RBT5_STANDARD_WELD_DATA : WORD ;
    RBT6_STANDARD_WELD_DATA : WORD ;
    RBT7_STANDARD_WELD_DATA : WORD ;
    RBT8_STANDARD_WELD_DATA : WORD ;
    RBT9_STANDARD_WELD_DATA : WORD ;
    RBT10_STANDARD_WELD_DATA : WORD ;
    RBT11_STANDARD_WELD_DATA : WORD ;
    RBT12_STANDARD_WELD_DATA : WORD ;
    RBT13_STANDARD_WELD_DATA : WORD ;
    RBT14_STANDARD_WELD_DATA : WORD ;
    RBT15_STANDARD_WELD_DATA : WORD ;
    RBT16_STANDARD_WELD_DATA : WORD ;
    RBT17_STANDARD_WELD_DATA : WORD ;
    RBT18_STANDARD_WELD_DATA : WORD ;
    RBT19_STANDARD_WELD_DATA : WORD ;
    RBT20_STANDARD_WELD_DATA : WORD ;
    RBT21_STANDARD_WELD_DATA : WORD ;
    RBT22_STANDARD_WELD_DATA : WORD ;
    RBT23_STANDARD_WELD_DAT : WORD ;
    RBT24_STANDARD_WELD_DAT : WORD ;
    CHK_WORD : WORD ;
    TEST_TEMP : ARRAY  [1 .. 40 ] OF BYTE ;
   END_STRUCT ;
   S702_BT_CODE_2113 : STRUCT
    STATION_MAIN : WORD ;
    DISTINCTION_LH_RH : WORD ;
    STAION_NUMBER : WORD ;
    BODY_TYPE_1ST : WORD ;
    BODY_TYPE_OPTION : WORD ;
    RBT1_STANDARD_WELD_DATA : WORD ;
    RBT2_STANDARD_WELD_DATA : WORD ;
    RBT3_STANDARD_WELD_DATA : WORD ;
    RBT4_STANDARD_WELD_DATA : WORD ;
    RBT5_STANDARD_WELD_DATA : WORD ;
    RBT6_STANDARD_WELD_DATA : WORD ;
    RBT7_STANDARD_WELD_DATA : WORD ;
    RBT8_STANDARD_WELD_DATA : WORD ;
    RBT9_STANDARD_WELD_DATA : WORD ;
    RBT10_STANDARD_WELD_DATA : WORD ;
    RBT11_STANDARD_WELD_DATA : WORD ;
    RBT12_STANDARD_WELD_DATA : WORD ;
    RBT13_STANDARD_WELD_DATA : WORD ;
    RBT14_STANDARD_WELD_DATA : WORD ;
    RBT15_STANDARD_WELD_DATA : WORD ;
    RBT16_STANDARD_WELD_DATA : WORD ;
    RBT17_STANDARD_WELD_DATA : WORD ;
    RBT18_STANDARD_WELD_DATA : WORD ;
    RBT19_STANDARD_WELD_DATA : WORD ;
    RBT20_STANDARD_WELD_DATA : WORD ;
    RBT21_STANDARD_WELD_DATA : WORD ;
    RBT22_STANDARD_WELD_DATA : WORD ;
    RBT23_STANDARD_WELD_DAT : WORD ;
    RBT24_STANDARD_WELD_DAT : WORD ;
    CHK_WORD : WORD ;
    TEST_TEMP : ARRAY  [1 .. 40 ] OF BYTE ;
   END_STRUCT ;
   S702_BT_CODE_2114 : STRUCT
    STATION_MAIN : WORD ;
    DISTINCTION_LH_RH : WORD ;
    STAION_NUMBER : WORD ;
    BODY_TYPE_1ST : WORD ;
    BODY_TYPE_OPTION : WORD ;
    RBT1_STANDARD_WELD_DATA : WORD ;
    RBT2_STANDARD_WELD_DATA : WORD ;
    RBT3_STANDARD_WELD_DATA : WORD ;
    RBT4_STANDARD_WELD_DATA : WORD ;
    RBT5_STANDARD_WELD_DATA : WORD ;
    RBT6_STANDARD_WELD_DATA : WORD ;
    RBT7_STANDARD_WELD_DATA : WORD ;
    RBT8_STANDARD_WELD_DATA : WORD ;
    RBT9_STANDARD_WELD_DATA : WORD ;
    RBT10_STANDARD_WELD_DATA : WORD ;
    RBT11_STANDARD_WELD_DATA : WORD ;
    RBT12_STANDARD_WELD_DATA : WORD ;
    RBT13_STANDARD_WELD_DATA : WORD ;
    RBT14_STANDARD_WELD_DATA : WORD ;
    RBT15_STANDARD_WELD_DATA : WORD ;
    RBT16_STANDARD_WELD_DATA : WORD ;
    RBT17_STANDARD_WELD_DATA : WORD ;
    RBT18_STANDARD_WELD_DATA : WORD ;
    RBT19_STANDARD_WELD_DATA : WORD ;
    RBT20_STANDARD_WELD_DATA : WORD ;
    RBT21_STANDARD_WELD_DATA : WORD ;
    RBT22_STANDARD_WELD_DATA : WORD ;
    RBT23_STANDARD_WELD_DAT : WORD ;
    RBT24_STANDARD_WELD_DAT : WORD ;
    CHK_WORD : WORD ;
    TEST_TEMP : ARRAY  [1 .. 40 ] OF BYTE ;
   END_STRUCT ;
   S702_BT_CODE_2115 : STRUCT
    STATION_MAIN : WORD ;
    DISTINCTION_LH_RH : WORD ;
    STAION_NUMBER : WORD ;
    BODY_TYPE_1ST : WORD ;
    BODY_TYPE_OPTION : WORD ;
    RBT1_STANDARD_WELD_DATA : WORD ;
    RBT2_STANDARD_WELD_DATA : WORD ;
    RBT3_STANDARD_WELD_DATA : WORD ;
    RBT4_STANDARD_WELD_DATA : WORD ;
    RBT5_STANDARD_WELD_DATA : WORD ;
    RBT6_STANDARD_WELD_DATA : WORD ;
    RBT7_STANDARD_WELD_DATA : WORD ;
    RBT8_STANDARD_WELD_DATA : WORD ;
    RBT9_STANDARD_WELD_DATA : WORD ;
    RBT10_STANDARD_WELD_DATA : WORD ;
    RBT11_STANDARD_WELD_DATA : WORD ;
    RBT12_STANDARD_WELD_DATA : WORD ;
    RBT13_STANDARD_WELD_DATA : WORD ;
    RBT14_STANDARD_WELD_DATA : WORD ;
    RBT15_STANDARD_WELD_DATA : WORD ;
    RBT16_STANDARD_WELD_DATA : WORD ;
    RBT17_STANDARD_WELD_DATA : WORD ;
    RBT18_STANDARD_WELD_DATA : WORD ;
    RBT19_STANDARD_WELD_DATA : WORD ;
    RBT20_STANDARD_WELD_DATA : WORD ;
    RBT21_STANDARD_WELD_DATA : WORD ;
    RBT22_STANDARD_WELD_DATA : WORD ;
    RBT23_STANDARD_WELD_DAT : WORD ;
    RBT24_STANDARD_WELD_DAT : WORD ;
    CHK_WORD : WORD ;
    TEST_TEMP : ARRAY  [1 .. 40 ] OF BYTE ;
   END_STRUCT ;
   S702_BT_CODE_2116 : STRUCT
    STATION_MAIN : WORD ;
    DISTINCTION_LH_RH : WORD ;
    STAION_NUMBER : WORD ;
    BODY_TYPE_1ST : WORD ;
    BODY_TYPE_OPTION : WORD ;
    RBT1_STANDARD_WELD_DATA : WORD ;
    RBT2_STANDARD_WELD_DATA : WORD ;
    RBT3_STANDARD_WELD_DATA : WORD ;
    RBT4_STANDARD_WELD_DATA : WORD ;
    RBT5_STANDARD_WELD_DATA : WORD ;
    RBT6_STANDARD_WELD_DATA : WORD ;
    RBT7_STANDARD_WELD_DATA : WORD ;
    RBT8_STANDARD_WELD_DATA : WORD ;
    RBT9_STANDARD_WELD_DATA : WORD ;
    RBT10_STANDARD_WELD_DATA : WORD ;
    RBT11_STANDARD_WELD_DATA : WORD ;
    RBT12_STANDARD_WELD_DATA : WORD ;
    RBT13_STANDARD_WELD_DATA : WORD ;
    RBT14_STANDARD_WELD_DATA : WORD ;
    RBT15_STANDARD_WELD_DATA : WORD ;
    RBT16_STANDARD_WELD_DATA : WORD ;
    RBT17_STANDARD_WELD_DATA : WORD ;
    RBT18_STANDARD_WELD_DATA : WORD ;
    RBT19_STANDARD_WELD_DATA : WORD ;
    RBT20_STANDARD_WELD_DATA : WORD ;
    RBT21_STANDARD_WELD_DATA : WORD ;
    RBT22_STANDARD_WELD_DATA : WORD ;
    RBT23_STANDARD_WELD_DAT : WORD ;
    RBT24_STANDARD_WELD_DAT : WORD ;
    CHK_WORD : WORD ;
    TEST_TEMP : ARRAY  [1 .. 40 ] OF BYTE ;
   END_STRUCT ;
   S702_BT_CODE_2117 : STRUCT
    STATION_MAIN : WORD ;
    DISTINCTION_LH_RH : WORD ;
    STAION_NUMBER : WORD ;
    BODY_TYPE_1ST : WORD ;
    BODY_TYPE_OPTION : WORD ;
    RBT1_STANDARD_WELD_DATA : WORD ;
    RBT2_STANDARD_WELD_DATA : WORD ;
    RBT3_STANDARD_WELD_DATA : WORD ;
    RBT4_STANDARD_WELD_DATA : WORD ;
    RBT5_STANDARD_WELD_DATA : WORD ;
    RBT6_STANDARD_WELD_DATA : WORD ;
    RBT7_STANDARD_WELD_DATA : WORD ;
    RBT8_STANDARD_WELD_DATA : WORD ;
    RBT9_STANDARD_WELD_DATA : WORD ;
    RBT10_STANDARD_WELD_DATA : WORD ;
    RBT11_STANDARD_WELD_DATA : WORD ;
    RBT12_STANDARD_WELD_DATA : WORD ;
    RBT13_STANDARD_WELD_DATA : WORD ;
    RBT14_STANDARD_WELD_DATA : WORD ;
    RBT15_STANDARD_WELD_DATA : WORD ;
    RBT16_STANDARD_WELD_DATA : WORD ;
    RBT17_STANDARD_WELD_DATA : WORD ;
    RBT18_STANDARD_WELD_DATA : WORD ;
    RBT19_STANDARD_WELD_DATA : WORD ;
    RBT20_STANDARD_WELD_DATA : WORD ;
    RBT21_STANDARD_WELD_DATA : WORD ;
    RBT22_STANDARD_WELD_DATA : WORD ;
    RBT23_STANDARD_WELD_DAT : WORD ;
    RBT24_STANDARD_WELD_DAT : WORD ;
    CHK_WORD : WORD ;
    TEST_TEMP : ARRAY  [1 .. 40 ] OF BYTE ;
   END_STRUCT ;
   S702_BT_CODE_2118 : STRUCT
    STATION_MAIN : WORD ;
    DISTINCTION_LH_RH : WORD ;
    STAION_NUMBER : WORD ;
    BODY_TYPE_1ST : WORD ;
    BODY_TYPE_OPTION : WORD ;
    RBT1_STANDARD_WELD_DATA : WORD ;
    RBT2_STANDARD_WELD_DATA : WORD ;
    RBT3_STANDARD_WELD_DATA : WORD ;
    RBT4_STANDARD_WELD_DATA : WORD ;
    RBT5_STANDARD_WELD_DATA : WORD ;
    RBT6_STANDARD_WELD_DATA : WORD ;
    RBT7_STANDARD_WELD_DATA : WORD ;
    RBT8_STANDARD_WELD_DATA : WORD ;
    RBT9_STANDARD_WELD_DATA : WORD ;
    RBT10_STANDARD_WELD_DATA : WORD ;
    RBT11_STANDARD_WELD_DATA : WORD ;
    RBT12_STANDARD_WELD_DATA : WORD ;
    RBT13_STANDARD_WELD_DATA : WORD ;
    RBT14_STANDARD_WELD_DATA : WORD ;
    RBT15_STANDARD_WELD_DATA : WORD ;
    RBT16_STANDARD_WELD_DATA : WORD ;
    RBT17_STANDARD_WELD_DATA : WORD ;
    RBT18_STANDARD_WELD_DATA : WORD ;
    RBT19_STANDARD_WELD_DATA : WORD ;
    RBT20_STANDARD_WELD_DATA : WORD ;
    RBT21_STANDARD_WELD_DATA : WORD ;
    RBT22_STANDARD_WELD_DATA : WORD ;
    RBT23_STANDARD_WELD_DAT : WORD ;
    RBT24_STANDARD_WELD_DAT : WORD ;
    CHK_WORD : WORD ;
    TEST_TEMP : ARRAY  [1 .. 40 ] OF BYTE ;
   END_STRUCT ;
   S702_BT_CODE_2119 : STRUCT
    STATION_MAIN : WORD ;
    DISTINCTION_LH_RH : WORD ;
    STAION_NUMBER : WORD ;
    BODY_TYPE_1ST : WORD ;
    BODY_TYPE_OPTION : WORD ;
    RBT1_STANDARD_WELD_DATA : WORD ;
    RBT2_STANDARD_WELD_DATA : WORD ;
    RBT3_STANDARD_WELD_DATA : WORD ;
    RBT4_STANDARD_WELD_DATA : WORD ;
    RBT5_STANDARD_WELD_DATA : WORD ;
    RBT6_STANDARD_WELD_DATA : WORD ;
    RBT7_STANDARD_WELD_DATA : WORD ;
    RBT8_STANDARD_WELD_DATA : WORD ;
    RBT9_STANDARD_WELD_DATA : WORD ;
    RBT10_STANDARD_WELD_DATA : WORD ;
    RBT11_STANDARD_WELD_DATA : WORD ;
    RBT12_STANDARD_WELD_DATA : WORD ;
    RBT13_STANDARD_WELD_DATA : WORD ;
    RBT14_STANDARD_WELD_DATA : WORD ;
    RBT15_STANDARD_WELD_DATA : WORD ;
    RBT16_STANDARD_WELD_DATA : WORD ;
    RBT17_STANDARD_WELD_DATA : WORD ;
    RBT18_STANDARD_WELD_DATA : WORD ;
    RBT19_STANDARD_WELD_DATA : WORD ;
    RBT20_STANDARD_WELD_DATA : WORD ;
    RBT21_STANDARD_WELD_DATA : WORD ;
    RBT22_STANDARD_WELD_DATA : WORD ;
    RBT23_STANDARD_WELD_DAT : WORD ;
    RBT24_STANDARD_WELD_DAT : WORD ;
    CHK_WORD : WORD ;
    TEST_TEMP : ARRAY  [1 .. 40 ] OF BYTE ;
   END_STRUCT ;
   S702_BT_CODE_2120 : STRUCT
    STATION_MAIN : WORD ;
    DISTINCTION_LH_RH : WORD ;
    STAION_NUMBER : WORD ;
    BODY_TYPE_1ST : WORD ;
    BODY_TYPE_OPTION : WORD ;
    RBT1_STANDARD_WELD_DATA : WORD ;
    RBT2_STANDARD_WELD_DATA : WORD ;
    RBT3_STANDARD_WELD_DATA : WORD ;
    RBT4_STANDARD_WELD_DATA : WORD ;
    RBT5_STANDARD_WELD_DATA : WORD ;
    RBT6_STANDARD_WELD_DATA : WORD ;
    RBT7_STANDARD_WELD_DATA : WORD ;
    RBT8_STANDARD_WELD_DATA : WORD ;
    RBT9_STANDARD_WELD_DATA : WORD ;
    RBT10_STANDARD_WELD_DATA : WORD ;
    RBT11_STANDARD_WELD_DATA : WORD ;
    RBT12_STANDARD_WELD_DATA : WORD ;
    RBT13_STANDARD_WELD_DATA : WORD ;
    RBT14_STANDARD_WELD_DATA : WORD ;
    RBT15_STANDARD_WELD_DATA : WORD ;
    RBT16_STANDARD_WELD_DATA : WORD ;
    RBT17_STANDARD_WELD_DATA : WORD ;
    RBT18_STANDARD_WELD_DATA : WORD ;
    RBT19_STANDARD_WELD_DATA : WORD ;
    RBT20_STANDARD_WELD_DATA : WORD ;
    RBT21_STANDARD_WELD_DATA : WORD ;
    RBT22_STANDARD_WELD_DATA : WORD ;
    RBT23_STANDARD_WELD_DAT : WORD ;
    RBT24_STANDARD_WELD_DAT : WORD ;
    CHK_WORD : WORD ;
    TEST_TEMP : ARRAY  [1 .. 40 ] OF BYTE ;
   END_STRUCT ;
   S704_BT_CODE_2101 : STRUCT
    STATION_MAIN : WORD ;
    DISTINCTION_LH_RH : WORD ;
    STAION_NUMBER : WORD ;
    BODY_TYPE_1ST : WORD ;
    BODY_TYPE_OPTION : WORD ;
    RBT1_STANDARD_WELD_DATA : WORD ;
    RBT2_STANDARD_WELD_DATA : WORD ;
    RBT3_STANDARD_WELD_DATA : WORD ;
    RBT4_STANDARD_WELD_DATA : WORD ;
    RBT5_STANDARD_WELD_DATA : WORD ;
    RBT6_STANDARD_WELD_DATA : WORD ;
    RBT7_STANDARD_WELD_DATA : WORD ;
    RBT8_STANDARD_WELD_DATA : WORD ;
    RBT9_STANDARD_WELD_DATA : WORD ;
    RBT10_STANDARD_WELD_DATA : WORD ;
    RBT11_STANDARD_WELD_DATA : WORD ;
    RBT12_STANDARD_WELD_DATA : WORD ;
    RBT13_STANDARD_WELD_DATA : WORD ;
    RBT14_STANDARD_WELD_DATA : WORD ;
    RBT15_STANDARD_WELD_DATA : WORD ;
    RBT16_STANDARD_WELD_DATA : WORD ;
    RBT17_STANDARD_WELD_DATA : WORD ;
    RBT18_STANDARD_WELD_DATA : WORD ;
    RBT19_STANDARD_WELD_DATA : WORD ;
    RBT20_STANDARD_WELD_DATA : WORD ;
    RBT21_STANDARD_WELD_DATA : WORD ;
    RBT22_STANDARD_WELD_DATA : WORD ;
    RBT23_STANDARD_WELD_DAT : WORD ;
    RBT24_STANDARD_WELD_DAT : WORD ;
    CHK_WORD : WORD ;
    TEST_TEMP : ARRAY  [1 .. 40 ] OF BYTE ;
   END_STRUCT ;
   S704_BT_CODE_2102 : STRUCT
    STATION_MAIN : WORD ;
    DISTINCTION_LH_RH : WORD ;
    STAION_NUMBER : WORD ;
    BODY_TYPE_1ST : WORD ;
    BODY_TYPE_OPTION : WORD ;
    RBT1_STANDARD_WELD_DATA : WORD ;
    RBT2_STANDARD_WELD_DATA : WORD ;
    RBT3_STANDARD_WELD_DATA : WORD ;
    RBT4_STANDARD_WELD_DATA : WORD ;
    RBT5_STANDARD_WELD_DATA : WORD ;
    RBT6_STANDARD_WELD_DATA : WORD ;
    RBT7_STANDARD_WELD_DATA : WORD ;
    RBT8_STANDARD_WELD_DATA : WORD ;
    RBT9_STANDARD_WELD_DATA : WORD ;
    RBT10_STANDARD_WELD_DATA : WORD ;
    RBT11_STANDARD_WELD_DATA : WORD ;
    RBT12_STANDARD_WELD_DATA : WORD ;
    RBT13_STANDARD_WELD_DATA : WORD ;
    RBT14_STANDARD_WELD_DATA : WORD ;
    RBT15_STANDARD_WELD_DATA : WORD ;
    RBT16_STANDARD_WELD_DATA : WORD ;
    RBT17_STANDARD_WELD_DATA : WORD ;
    RBT18_STANDARD_WELD_DATA : WORD ;
    RBT19_STANDARD_WELD_DATA : WORD ;
    RBT20_STANDARD_WELD_DATA : WORD ;
    RBT21_STANDARD_WELD_DATA : WORD ;
    RBT22_STANDARD_WELD_DATA : WORD ;
    RBT23_STANDARD_WELD_DAT : WORD ;
    RBT24_STANDARD_WELD_DAT : WORD ;
    CHK_WORD : WORD ;
    TEST_TEMP : ARRAY  [1 .. 40 ] OF BYTE ;
   END_STRUCT ;
   S704_BT_CODE_2103 : STRUCT
    STATION_MAIN : WORD ;
    DISTINCTION_LH_RH : WORD ;
    STAION_NUMBER : WORD ;
    BODY_TYPE_1ST : WORD ;
    BODY_TYPE_OPTION : WORD ;
    RBT1_STANDARD_WELD_DATA : WORD ;
    RBT2_STANDARD_WELD_DATA : WORD ;
    RBT3_STANDARD_WELD_DATA : WORD ;
    RBT4_STANDARD_WELD_DATA : WORD ;
    RBT5_STANDARD_WELD_DATA : WORD ;
    RBT6_STANDARD_WELD_DATA : WORD ;
    RBT7_STANDARD_WELD_DATA : WORD ;
    RBT8_STANDARD_WELD_DATA : WORD ;
    RBT9_STANDARD_WELD_DATA : WORD ;
    RBT10_STANDARD_WELD_DATA : WORD ;
    RBT11_STANDARD_WELD_DATA : WORD ;
    RBT12_STANDARD_WELD_DATA : WORD ;
    RBT13_STANDARD_WELD_DATA : WORD ;
    RBT14_STANDARD_WELD_DATA : WORD ;
    RBT15_STANDARD_WELD_DATA : WORD ;
    RBT16_STANDARD_WELD_DATA : WORD ;
    RBT17_STANDARD_WELD_DATA : WORD ;
    RBT18_STANDARD_WELD_DATA : WORD ;
    RBT19_STANDARD_WELD_DATA : WORD ;
    RBT20_STANDARD_WELD_DATA : WORD ;
    RBT21_STANDARD_WELD_DATA : WORD ;
    RBT22_STANDARD_WELD_DATA : WORD ;
    RBT23_STANDARD_WELD_DAT : WORD ;
    RBT24_STANDARD_WELD_DAT : WORD ;
    CHK_WORD : WORD ;
    TEST_TEMP : ARRAY  [1 .. 40 ] OF BYTE ;
   END_STRUCT ;
   S704_BT_CODE_2104 : STRUCT
    STATION_MAIN : WORD ;
    DISTINCTION_LH_RH : WORD ;
    STAION_NUMBER : WORD ;
    BODY_TYPE_1ST : WORD ;
    BODY_TYPE_OPTION : WORD ;
    RBT1_STANDARD_WELD_DATA : WORD ;
    RBT2_STANDARD_WELD_DATA : WORD ;
    RBT3_STANDARD_WELD_DATA : WORD ;
    RBT4_STANDARD_WELD_DATA : WORD ;
    RBT5_STANDARD_WELD_DATA : WORD ;
    RBT6_STANDARD_WELD_DATA : WORD ;
    RBT7_STANDARD_WELD_DATA : WORD ;
    RBT8_STANDARD_WELD_DATA : WORD ;
    RBT9_STANDARD_WELD_DATA : WORD ;
    RBT10_STANDARD_WELD_DATA : WORD ;
    RBT11_STANDARD_WELD_DATA : WORD ;
    RBT12_STANDARD_WELD_DATA : WORD ;
    RBT13_STANDARD_WELD_DATA : WORD ;
    RBT14_STANDARD_WELD_DATA : WORD ;
    RBT15_STANDARD_WELD_DATA : WORD ;
    RBT16_STANDARD_WELD_DATA : WORD ;
    RBT17_STANDARD_WELD_DATA : WORD ;
    RBT18_STANDARD_WELD_DATA : WORD ;
    RBT19_STANDARD_WELD_DATA : WORD ;
    RBT20_STANDARD_WELD_DATA : WORD ;
    RBT21_STANDARD_WELD_DATA : WORD ;
    RBT22_STANDARD_WELD_DATA : WORD ;
    RBT23_STANDARD_WELD_DAT : WORD ;
    RBT24_STANDARD_WELD_DAT : WORD ;
    CHK_WORD : WORD ;
    TEST_TEMP : ARRAY  [1 .. 40 ] OF BYTE ;
   END_STRUCT ;
   S704_BT_CODE_2105 : STRUCT
    STATION_MAIN : WORD ;
    DISTINCTION_LH_RH : WORD ;
    STAION_NUMBER : WORD ;
    BODY_TYPE_1ST : WORD ;
    BODY_TYPE_OPTION : WORD ;
    RBT1_STANDARD_WELD_DATA : WORD ;
    RBT2_STANDARD_WELD_DATA : WORD ;
    RBT3_STANDARD_WELD_DATA : WORD ;
    RBT4_STANDARD_WELD_DATA : WORD ;
    RBT5_STANDARD_WELD_DATA : WORD ;
    RBT6_STANDARD_WELD_DATA : WORD ;
    RBT7_STANDARD_WELD_DATA : WORD ;
    RBT8_STANDARD_WELD_DATA : WORD ;
    RBT9_STANDARD_WELD_DATA : WORD ;
    RBT10_STANDARD_WELD_DATA : WORD ;
    RBT11_STANDARD_WELD_DATA : WORD ;
    RBT12_STANDARD_WELD_DATA : WORD ;
    RBT13_STANDARD_WELD_DATA : WORD ;
    RBT14_STANDARD_WELD_DATA : WORD ;
    RBT15_STANDARD_WELD_DATA : WORD ;
    RBT16_STANDARD_WELD_DATA : WORD ;
    RBT17_STANDARD_WELD_DATA : WORD ;
    RBT18_STANDARD_WELD_DATA : WORD ;
    RBT19_STANDARD_WELD_DATA : WORD ;
    RBT20_STANDARD_WELD_DATA : WORD ;
    RBT21_STANDARD_WELD_DATA : WORD ;
    RBT22_STANDARD_WELD_DATA : WORD ;
    RBT23_STANDARD_WELD_DAT : WORD ;
    RBT24_STANDARD_WELD_DAT : WORD ;
    CHK_WORD : WORD ;
    TEST_TEMP : ARRAY  [1 .. 40 ] OF BYTE ;
   END_STRUCT ;
   S704_BT_CODE_2106 : STRUCT
    STATION_MAIN : WORD ;
    DISTINCTION_LH_RH : WORD ;
    STAION_NUMBER : WORD ;
    BODY_TYPE_1ST : WORD ;
    BODY_TYPE_OPTION : WORD ;
    RBT1_STANDARD_WELD_DATA : WORD ;
    RBT2_STANDARD_WELD_DATA : WORD ;
    RBT3_STANDARD_WELD_DATA : WORD ;
    RBT4_STANDARD_WELD_DATA : WORD ;
    RBT5_STANDARD_WELD_DATA : WORD ;
    RBT6_STANDARD_WELD_DATA : WORD ;
    RBT7_STANDARD_WELD_DATA : WORD ;
    RBT8_STANDARD_WELD_DATA : WORD ;
    RBT9_STANDARD_WELD_DATA : WORD ;
    RBT10_STANDARD_WELD_DATA : WORD ;
    RBT11_STANDARD_WELD_DATA : WORD ;
    RBT12_STANDARD_WELD_DATA : WORD ;
    RBT13_STANDARD_WELD_DATA : WORD ;
    RBT14_STANDARD_WELD_DATA : WORD ;
    RBT15_STANDARD_WELD_DATA : WORD ;
    RBT16_STANDARD_WELD_DATA : WORD ;
    RBT17_STANDARD_WELD_DATA : WORD ;
    RBT18_STANDARD_WELD_DATA : WORD ;
    RBT19_STANDARD_WELD_DATA : WORD ;
    RBT20_STANDARD_WELD_DATA : WORD ;
    RBT21_STANDARD_WELD_DATA : WORD ;
    RBT22_STANDARD_WELD_DATA : WORD ;
    RBT23_STANDARD_WELD_DAT : WORD ;
    RBT24_STANDARD_WELD_DAT : WORD ;
    CHK_WORD : WORD ;
    TEST_TEMP : ARRAY  [1 .. 40 ] OF BYTE ;
   END_STRUCT ;
   S704_BT_CODE_2107 : STRUCT
    STATION_MAIN : WORD ;
    DISTINCTION_LH_RH : WORD ;
    STAION_NUMBER : WORD ;
    BODY_TYPE_1ST : WORD ;
    BODY_TYPE_OPTION : WORD ;
    RBT1_STANDARD_WELD_DATA : WORD ;
    RBT2_STANDARD_WELD_DATA : WORD ;
    RBT3_STANDARD_WELD_DATA : WORD ;
    RBT4_STANDARD_WELD_DATA : WORD ;
    RBT5_STANDARD_WELD_DATA : WORD ;
    RBT6_STANDARD_WELD_DATA : WORD ;
    RBT7_STANDARD_WELD_DATA : WORD ;
    RBT8_STANDARD_WELD_DATA : WORD ;
    RBT9_STANDARD_WELD_DATA : WORD ;
    RBT10_STANDARD_WELD_DATA : WORD ;
    RBT11_STANDARD_WELD_DATA : WORD ;
    RBT12_STANDARD_WELD_DATA : WORD ;
    RBT13_STANDARD_WELD_DATA : WORD ;
    RBT14_STANDARD_WELD_DATA : WORD ;
    RBT15_STANDARD_WELD_DATA : WORD ;
    RBT16_STANDARD_WELD_DATA : WORD ;
    RBT17_STANDARD_WELD_DATA : WORD ;
    RBT18_STANDARD_WELD_DATA : WORD ;
    RBT19_STANDARD_WELD_DATA : WORD ;
    RBT20_STANDARD_WELD_DATA : WORD ;
    RBT21_STANDARD_WELD_DATA : WORD ;
    RBT22_STANDARD_WELD_DATA : WORD ;
    RBT23_STANDARD_WELD_DAT : WORD ;
    RBT24_STANDARD_WELD_DAT : WORD ;
    CHK_WORD : WORD ;
    TEST_TEMP : ARRAY  [1 .. 40 ] OF BYTE ;
   END_STRUCT ;
   S704_BT_CODE_2108 : STRUCT
    STATION_MAIN : WORD ;
    DISTINCTION_LH_RH : WORD ;
    STAION_NUMBER : WORD ;
    BODY_TYPE_1ST : WORD ;
    BODY_TYPE_OPTION : WORD ;
    RBT1_STANDARD_WELD_DATA : WORD ;
    RBT2_STANDARD_WELD_DATA : WORD ;
    RBT3_STANDARD_WELD_DATA : WORD ;
    RBT4_STANDARD_WELD_DATA : WORD ;
    RBT5_STANDARD_WELD_DATA : WORD ;
    RBT6_STANDARD_WELD_DATA : WORD ;
    RBT7_STANDARD_WELD_DATA : WORD ;
    RBT8_STANDARD_WELD_DATA : WORD ;
    RBT9_STANDARD_WELD_DATA : WORD ;
    RBT10_STANDARD_WELD_DATA : WORD ;
    RBT11_STANDARD_WELD_DATA : WORD ;
    RBT12_STANDARD_WELD_DATA : WORD ;
    RBT13_STANDARD_WELD_DATA : WORD ;
    RBT14_STANDARD_WELD_DATA : WORD ;
    RBT15_STANDARD_WELD_DATA : WORD ;
    RBT16_STANDARD_WELD_DATA : WORD ;
    RBT17_STANDARD_WELD_DATA : WORD ;
    RBT18_STANDARD_WELD_DATA : WORD ;
    RBT19_STANDARD_WELD_DATA : WORD ;
    RBT20_STANDARD_WELD_DATA : WORD ;
    RBT21_STANDARD_WELD_DATA : WORD ;
    RBT22_STANDARD_WELD_DATA : WORD ;
    RBT23_STANDARD_WELD_DAT : WORD ;
    RBT24_STANDARD_WELD_DAT : WORD ;
    CHK_WORD : WORD ;
    TEST_TEMP : ARRAY  [1 .. 40 ] OF BYTE ;
   END_STRUCT ;
   S704_BT_CODE_2109 : STRUCT
    STATION_MAIN : WORD ;
    DISTINCTION_LH_RH : WORD ;
    STAION_NUMBER : WORD ;
    BODY_TYPE_1ST : WORD ;
    BODY_TYPE_OPTION : WORD ;
    RBT1_STANDARD_WELD_DATA : WORD ;
    RBT2_STANDARD_WELD_DATA : WORD ;
    RBT3_STANDARD_WELD_DATA : WORD ;
    RBT4_STANDARD_WELD_DATA : WORD ;
    RBT5_STANDARD_WELD_DATA : WORD ;
    RBT6_STANDARD_WELD_DATA : WORD ;
    RBT7_STANDARD_WELD_DATA : WORD ;
    RBT8_STANDARD_WELD_DATA : WORD ;
    RBT9_STANDARD_WELD_DATA : WORD ;
    RBT10_STANDARD_WELD_DATA : WORD ;
    RBT11_STANDARD_WELD_DATA : WORD ;
    RBT12_STANDARD_WELD_DATA : WORD ;
    RBT13_STANDARD_WELD_DATA : WORD ;
    RBT14_STANDARD_WELD_DATA : WORD ;
    RBT15_STANDARD_WELD_DATA : WORD ;
    RBT16_STANDARD_WELD_DATA : WORD ;
    RBT17_STANDARD_WELD_DATA : WORD ;
    RBT18_STANDARD_WELD_DATA : WORD ;
    RBT19_STANDARD_WELD_DATA : WORD ;
    RBT20_STANDARD_WELD_DATA : WORD ;
    RBT21_STANDARD_WELD_DATA : WORD ;
    RBT22_STANDARD_WELD_DATA : WORD ;
    RBT23_STANDARD_WELD_DAT : WORD ;
    RBT24_STANDARD_WELD_DAT : WORD ;
    CHK_WORD : WORD ;
    TEST_TEMP : ARRAY  [1 .. 40 ] OF BYTE ;
   END_STRUCT ;
   S704_BT_CODE_2110 : STRUCT
    STATION_MAIN : WORD ;
    DISTINCTION_LH_RH : WORD ;
    STAION_NUMBER : WORD ;
    BODY_TYPE_1ST : WORD ;
    BODY_TYPE_OPTION : WORD ;
    RBT1_STANDARD_WELD_DATA : WORD ;
    RBT2_STANDARD_WELD_DATA : WORD ;
    RBT3_STANDARD_WELD_DATA : WORD ;
    RBT4_STANDARD_WELD_DATA : WORD ;
    RBT5_STANDARD_WELD_DATA : WORD ;
    RBT6_STANDARD_WELD_DATA : WORD ;
    RBT7_STANDARD_WELD_DATA : WORD ;
    RBT8_STANDARD_WELD_DATA : WORD ;
    RBT9_STANDARD_WELD_DATA : WORD ;
    RBT10_STANDARD_WELD_DATA : WORD ;
    RBT11_STANDARD_WELD_DATA : WORD ;
    RBT12_STANDARD_WELD_DATA : WORD ;
    RBT13_STANDARD_WELD_DATA : WORD ;
    RBT14_STANDARD_WELD_DATA : WORD ;
    RBT15_STANDARD_WELD_DATA : WORD ;
    RBT16_STANDARD_WELD_DATA : WORD ;
    RBT17_STANDARD_WELD_DATA : WORD ;
    RBT18_STANDARD_WELD_DATA : WORD ;
    RBT19_STANDARD_WELD_DATA : WORD ;
    RBT20_STANDARD_WELD_DATA : WORD ;
    RBT21_STANDARD_WELD_DATA : WORD ;
    RBT22_STANDARD_WELD_DATA : WORD ;
    RBT23_STANDARD_WELD_DAT : WORD ;
    RBT24_STANDARD_WELD_DAT : WORD ;
    CHK_WORD : WORD ;
    TEST_TEMP : ARRAY  [1 .. 40 ] OF BYTE ;
   END_STRUCT ;
   S704_BT_CODE_2111 : STRUCT
    STATION_MAIN : WORD ;
    DISTINCTION_LH_RH : WORD ;
    STAION_NUMBER : WORD ;
    BODY_TYPE_1ST : WORD ;
    BODY_TYPE_OPTION : WORD ;
    RBT1_STANDARD_WELD_DATA : WORD ;
    RBT2_STANDARD_WELD_DATA : WORD ;
    RBT3_STANDARD_WELD_DATA : WORD ;
    RBT4_STANDARD_WELD_DATA : WORD ;
    RBT5_STANDARD_WELD_DATA : WORD ;
    RBT6_STANDARD_WELD_DATA : WORD ;
    RBT7_STANDARD_WELD_DATA : WORD ;
    RBT8_STANDARD_WELD_DATA : WORD ;
    RBT9_STANDARD_WELD_DATA : WORD ;
    RBT10_STANDARD_WELD_DATA : WORD ;
    RBT11_STANDARD_WELD_DATA : WORD ;
    RBT12_STANDARD_WELD_DATA : WORD ;
    RBT13_STANDARD_WELD_DATA : WORD ;
    RBT14_STANDARD_WELD_DATA : WORD ;
    RBT15_STANDARD_WELD_DATA : WORD ;
    RBT16_STANDARD_WELD_DATA : WORD ;
    RBT17_STANDARD_WELD_DATA : WORD ;
    RBT18_STANDARD_WELD_DATA : WORD ;
    RBT19_STANDARD_WELD_DATA : WORD ;
    RBT20_STANDARD_WELD_DATA : WORD ;
    RBT21_STANDARD_WELD_DATA : WORD ;
    RBT22_STANDARD_WELD_DATA : WORD ;
    RBT23_STANDARD_WELD_DAT : WORD ;
    RBT24_STANDARD_WELD_DAT : WORD ;
    CHK_WORD : WORD ;
    TEST_TEMP : ARRAY  [1 .. 40 ] OF BYTE ;
   END_STRUCT ;
   S704_BT_CODE_2112 : STRUCT
    STATION_MAIN : WORD ;
    DISTINCTION_LH_RH : WORD ;
    STAION_NUMBER : WORD ;
    BODY_TYPE_1ST : WORD ;
    BODY_TYPE_OPTION : WORD ;
    RBT1_STANDARD_WELD_DATA : WORD ;
    RBT2_STANDARD_WELD_DATA : WORD ;
    RBT3_STANDARD_WELD_DATA : WORD ;
    RBT4_STANDARD_WELD_DATA : WORD ;
    RBT5_STANDARD_WELD_DATA : WORD ;
    RBT6_STANDARD_WELD_DATA : WORD ;
    RBT7_STANDARD_WELD_DATA : WORD ;
    RBT8_STANDARD_WELD_DATA : WORD ;
    RBT9_STANDARD_WELD_DATA : WORD ;
    RBT10_STANDARD_WELD_DATA : WORD ;
    RBT11_STANDARD_WELD_DATA : WORD ;
    RBT12_STANDARD_WELD_DATA : WORD ;
    RBT13_STANDARD_WELD_DATA : WORD ;
    RBT14_STANDARD_WELD_DATA : WORD ;
    RBT15_STANDARD_WELD_DATA : WORD ;
    RBT16_STANDARD_WELD_DATA : WORD ;
    RBT17_STANDARD_WELD_DATA : WORD ;
    RBT18_STANDARD_WELD_DATA : WORD ;
    RBT19_STANDARD_WELD_DATA : WORD ;
    RBT20_STANDARD_WELD_DATA : WORD ;
    RBT21_STANDARD_WELD_DATA : WORD ;
    RBT22_STANDARD_WELD_DATA : WORD ;
    RBT23_STANDARD_WELD_DAT : WORD ;
    RBT24_STANDARD_WELD_DAT : WORD ;
    CHK_WORD : WORD ;
    TEST_TEMP : ARRAY  [1 .. 40 ] OF BYTE ;
   END_STRUCT ;
   S704_BT_CODE_2113 : STRUCT
    STATION_MAIN : WORD ;
    DISTINCTION_LH_RH : WORD ;
    STAION_NUMBER : WORD ;
    BODY_TYPE_1ST : WORD ;
    BODY_TYPE_OPTION : WORD ;
    RBT1_STANDARD_WELD_DATA : WORD ;
    RBT2_STANDARD_WELD_DATA : WORD ;
    RBT3_STANDARD_WELD_DATA : WORD ;
    RBT4_STANDARD_WELD_DATA : WORD ;
    RBT5_STANDARD_WELD_DATA : WORD ;
    RBT6_STANDARD_WELD_DATA : WORD ;
    RBT7_STANDARD_WELD_DATA : WORD ;
    RBT8_STANDARD_WELD_DATA : WORD ;
    RBT9_STANDARD_WELD_DATA : WORD ;
    RBT10_STANDARD_WELD_DATA : WORD ;
    RBT11_STANDARD_WELD_DATA : WORD ;
    RBT12_STANDARD_WELD_DATA : WORD ;
    RBT13_STANDARD_WELD_DATA : WORD ;
    RBT14_STANDARD_WELD_DATA : WORD ;
    RBT15_STANDARD_WELD_DATA : WORD ;
    RBT16_STANDARD_WELD_DATA : WORD ;
    RBT17_STANDARD_WELD_DATA : WORD ;
    RBT18_STANDARD_WELD_DATA : WORD ;
    RBT19_STANDARD_WELD_DATA : WORD ;
    RBT20_STANDARD_WELD_DATA : WORD ;
    RBT21_STANDARD_WELD_DATA : WORD ;
    RBT22_STANDARD_WELD_DATA : WORD ;
    RBT23_STANDARD_WELD_DAT : WORD ;
    RBT24_STANDARD_WELD_DAT : WORD ;
    CHK_WORD : WORD ;
    TEST_TEMP : ARRAY  [1 .. 40 ] OF BYTE ;
   END_STRUCT ;
   S704_BT_CODE_2114 : STRUCT
    STATION_MAIN : WORD ;
    DISTINCTION_LH_RH : WORD ;
    STAION_NUMBER : WORD ;
    BODY_TYPE_1ST : WORD ;
    BODY_TYPE_OPTION : WORD ;
    RBT1_STANDARD_WELD_DATA : WORD ;
    RBT2_STANDARD_WELD_DATA : WORD ;
    RBT3_STANDARD_WELD_DATA : WORD ;
    RBT4_STANDARD_WELD_DATA : WORD ;
    RBT5_STANDARD_WELD_DATA : WORD ;
    RBT6_STANDARD_WELD_DATA : WORD ;
    RBT7_STANDARD_WELD_DATA : WORD ;
    RBT8_STANDARD_WELD_DATA : WORD ;
    RBT9_STANDARD_WELD_DATA : WORD ;
    RBT10_STANDARD_WELD_DATA : WORD ;
    RBT11_STANDARD_WELD_DATA : WORD ;
    RBT12_STANDARD_WELD_DATA : WORD ;
    RBT13_STANDARD_WELD_DATA : WORD ;
    RBT14_STANDARD_WELD_DATA : WORD ;
    RBT15_STANDARD_WELD_DATA : WORD ;
    RBT16_STANDARD_WELD_DATA : WORD ;
    RBT17_STANDARD_WELD_DATA : WORD ;
    RBT18_STANDARD_WELD_DATA : WORD ;
    RBT19_STANDARD_WELD_DATA : WORD ;
    RBT20_STANDARD_WELD_DATA : WORD ;
    RBT21_STANDARD_WELD_DATA : WORD ;
    RBT22_STANDARD_WELD_DATA : WORD ;
    RBT23_STANDARD_WELD_DAT : WORD ;
    RBT24_STANDARD_WELD_DAT : WORD ;
    CHK_WORD : WORD ;
    TEST_TEMP : ARRAY  [1 .. 40 ] OF BYTE ;
   END_STRUCT ;
   S704_BT_CODE_2115 : STRUCT
    STATION_MAIN : WORD ;
    DISTINCTION_LH_RH : WORD ;
    STAION_NUMBER : WORD ;
    BODY_TYPE_1ST : WORD ;
    BODY_TYPE_OPTION : WORD ;
    RBT1_STANDARD_WELD_DATA : WORD ;
    RBT2_STANDARD_WELD_DATA : WORD ;
    RBT3_STANDARD_WELD_DATA : WORD ;
    RBT4_STANDARD_WELD_DATA : WORD ;
    RBT5_STANDARD_WELD_DATA : WORD ;
    RBT6_STANDARD_WELD_DATA : WORD ;
    RBT7_STANDARD_WELD_DATA : WORD ;
    RBT8_STANDARD_WELD_DATA : WORD ;
    RBT9_STANDARD_WELD_DATA : WORD ;
    RBT10_STANDARD_WELD_DATA : WORD ;
    RBT11_STANDARD_WELD_DATA : WORD ;
    RBT12_STANDARD_WELD_DATA : WORD ;
    RBT13_STANDARD_WELD_DATA : WORD ;
    RBT14_STANDARD_WELD_DATA : WORD ;
    RBT15_STANDARD_WELD_DATA : WORD ;
    RBT16_STANDARD_WELD_DATA : WORD ;
    RBT17_STANDARD_WELD_DATA : WORD ;
    RBT18_STANDARD_WELD_DATA : WORD ;
    RBT19_STANDARD_WELD_DATA : WORD ;
    RBT20_STANDARD_WELD_DATA : WORD ;
    RBT21_STANDARD_WELD_DATA : WORD ;
    RBT22_STANDARD_WELD_DATA : WORD ;
    RBT23_STANDARD_WELD_DAT : WORD ;
    RBT24_STANDARD_WELD_DAT : WORD ;
    CHK_WORD : WORD ;
    TEST_TEMP : ARRAY  [1 .. 40 ] OF BYTE ;
   END_STRUCT ;
   S704_BT_CODE_2116 : STRUCT
    STATION_MAIN : WORD ;
    DISTINCTION_LH_RH : WORD ;
    STAION_NUMBER : WORD ;
    BODY_TYPE_1ST : WORD ;
    BODY_TYPE_OPTION : WORD ;
    RBT1_STANDARD_WELD_DATA : WORD ;
    RBT2_STANDARD_WELD_DATA : WORD ;
    RBT3_STANDARD_WELD_DATA : WORD ;
    RBT4_STANDARD_WELD_DATA : WORD ;
